C05428=1039.258,123.258,-94.133,169.875,39.736,157.485
C05429=1039.265,123.507,-94.154,169.877,39.737,157.486
C05430=1039.270,123.756,-94.175,169.879,39.737,157.486
C05431=1039.276,124.006,-94.195,169.881,39.737,157.486
C05432=1039.283,124.254,-94.216,169.883,39.738,157.486
C05433=1039.289,124.504,-94.237,169.886,39.738,157.486
C05434=1039.296,124.789,-94.260,169.888,39.739,157.486
C05435=1039.303,125.075,-94.284,169.891,39.739,157.487
C05436=1039.310,125.362,-94.307,169.893,39.740,157.487
C05437=1039.317,125.647,-94.331,169.895,39.740,157.487
C05438=1039.324,125.896,-94.352,169.897,39.741,157.487
C05439=1039.330,126.145,-94.372,169.899,39.741,157.487
C05440=1039.336,126.394,-94.393,169.902,39.741,157.487
C05441=1039.343,126.643,-94.414,169.905,39.741,157.487
C05442=1039.349,126.892,-94.434,169.907,39.742,157.488
C05443=1039.355,127.141,-94.456,169.909,39.742,157.488
C05444=1039.361,127.390,-94.476,169.911,39.743,157.488
C05445=1039.368,127.639,-94.497,169.913,39.743,157.488
C05446=1039.373,127.889,-94.517,169.915,39.744,157.488
C05447=1039.379,128.138,-94.537,169.918,39.744,157.488
C05448=1039.386,128.387,-94.558,169.920,39.745,157.489
C05449=1039.392,128.636,-94.579,169.922,39.744,157.489
C05450=1039.399,128.885,-94.600,169.924,39.745,157.489
C05451=1039.405,129.134,-94.620,169.926,39.745,157.489
C05452=1039.411,129.383,-94.642,169.928,39.746,157.489
C05453=1039.417,129.632,-94.662,169.930,39.746,157.489
C05454=1039.424,129.881,-94.683,169.934,39.747,157.490
C05455=1039.429,130.130,-94.704,169.936,39.747,157.490
C05456=1039.436,130.379,-94.725,169.938,39.748,157.490
C05457=1039.442,130.628,-94.746,169.940,39.747,157.490
C05458=1039.448,130.877,-94.766,169.942,39.748,157.490
C05459=1039.455,131.126,-94.787,169.944,39.748,157.490
C05460=1039.461,131.376,-94.808,169.946,39.749,157.490
C05461=1039.467,131.624,-94.829,169.948,39.749,157.491
C05462=1039.474,131.873,-94.850,169.951,39.750,157.491
C05463=1039.480,132.123,-94.871,169.953,39.750,157.491
C05464=1039.485,132.372,-94.893,169.955,39.751,157.491
C05465=1039.492,132.620,-94.914,169.957,39.752,157.491
C05466=1039.497,132.870,-94.934,169.959,39.752,157.492
C05467=1039.503,133.119,-94.956,169.963,39.753,157.492
C05468=1039.510,133.368,-94.977,169.965,39.753,157.492
C05469=1039.516,133.617,-94.998,169.967,39.753,157.492
C05470=1039.522,133.866,-95.019,169.969,39.754,157.492
C05471=1039.529,134.115,-95.040,169.971,39.754,157.492
C05472=1039.534,134.363,-95.061,169.973,39.755,157.493
C05473=1039.540,134.613,-95.082,169.975,39.755,157.493
C05474=1039.547,134.862,-95.103,169.978,39.756,157.493
C05475=1039.553,135.111,-95.125,169.980,39.756,157.493
C05476=1039.559,135.360,-95.146,169.982,39.757,157.493
C05477=1039.565,135.609,-95.167,169.984,39.757,157.493
C05478=1039.571,135.859,-95.188,169.986,39.758,157.494
C05479=1039.577,136.107,-95.210,169.988,39.758,157.494
C05480=1039.584,136.356,-95.231,169.992,39.758,157.494
C05481=1039.590,136.605,-95.252,169.994,39.759,157.494
C05482=1039.595,136.854,-95.273,169.996,39.759,157.494
C05483=1039.602,137.103,-95.294,169.998,39.760,157.494
C05484=1039.608,137.352,-95.315,170.000,39.760,157.495
C05485=1039.615,137.602,-95.337,170.002,39.761,157.495
C05486=1039.620,137.850,-95.358,170.005,39.761,157.495
C05487=1039.627,138.099,-95.379,170.007,39.762,157.495
C05488=1039.633,138.348,-95.401,170.009,39.762,157.495
C05489=1039.639,138.597,-95.423,170.011,39.763,157.496
C05490=1039.645,138.846,-95.443,170.014,39.764,157.496
C05491=1039.652,139.095,-95.464,170.016,39.764,157.496
C05492=1039.658,139.345,-95.486,170.019,39.764,157.496
C05493=1039.663,139.593,-95.507,170.021,39.765,157.496
C05494=1039.669,139.842,-95.529,170.023,39.765,157.497
C05495=1039.676,140.091,-95.550,170.025,39.766,157.497
C05496=1039.682,140.341,-95.572,170.027,39.766,157.497
C05497=1039.687,140.589,-95.593,170.029,39.767,157.497
C05498=1039.695,140.875,-95.618,170.033,39.768,157.497
C05499=1039.701,141.160,-95.642,170.035,39.768,157.498
C05500=1039.709,141.446,-95.668,170.037,39.769,157.498
C05501=1039.716,141.731,-95.692,170.040,39.770,157.498
C05502=1039.722,141.980,-95.714,170.042,39.770,157.498
C05503=1039.728,142.229,-95.735,170.045,39.771,157.498
C05504=1039.734,142.479,-95.757,170.047,39.771,157.499
C05505=1039.741,142.728,-95.779,170.049,39.772,157.499
C05506=1039.746,142.976,-95.800,170.051,39.772,157.499
C05507=1039.752,143.225,-95.821,170.054,39.772,157.499
C05508=1039.759,143.475,-95.843,170.057,39.773,157.499
C05509=1039.765,143.724,-95.865,170.059,39.774,157.500
C05510=1039.771,143.973,-95.886,170.061,39.774,157.500
C05511=1039.776,144.222,-95.908,170.063,39.775,157.500
C05512=1039.783,144.470,-95.930,170.065,39.775,157.500
C05513=1039.789,144.719,-95.952,170.067,39.776,157.500
C05514=1039.795,144.969,-95.973,170.070,39.776,157.500
C05515=1039.802,145.217,-95.994,170.073,39.777,157.501
C05516=1039.808,145.467,-96.016,170.075,39.778,157.501
C05517=1039.814,145.715,-96.037,170.077,39.778,157.501
C05518=1039.820,145.964,-96.059,170.079,39.779,157.501
C05519=1039.826,146.213,-96.081,170.081,39.779,157.501
C05520=1039.833,146.462,-96.103,170.084,39.780,157.502
C05521=1039.839,146.711,-96.124,170.087,39.780,157.502
C05522=1039.845,146.961,-96.146,170.089,39.780,157.502
C05523=1039.851,147.209,-96.168,170.091,39.781,157.502
C05524=1039.858,147.458,-96.190,170.093,39.782,157.502
C05525=1039.863,147.707,-96.211,170.095,39.782,157.503
C05526=1039.869,147.956,-96.234,170.098,39.783,157.503
C05527=1039.875,148.205,-96.256,170.100,39.783,157.503
C05528=1039.881,148.454,-96.278,170.103,39.784,157.503
C05529=1039.887,148.703,-96.299,170.105,39.785,157.503
C05530=1039.894,148.952,-96.322,170.107,39.785,157.504
C05531=1039.900,149.201,-96.343,170.110,39.786,157.504
C05532=1039.906,149.450,-96.365,170.112,39.787,157.504
C05533=1039.912,149.698,-96.387,170.114,39.787,157.504
C05534=1039.917,149.948,-96.409,170.117,39.788,157.504
C05535=1039.924,150.197,-96.431,170.119,39.788,157.505
C05536=1039.930,150.446,-96.453,170.122,39.789,157.505
C05537=1039.936,150.695,-96.475,170.124,39.790,157.505
C05538=1039.942,150.944,-96.496,170.126,39.790,157.505
C05539=1039.948,151.193,-96.519,170.128,39.790,157.505
C05540=1039.954,151.442,-96.541,170.131,39.791,157.506
C05541=1039.961,151.691,-96.563,170.134,39.792,157.506
C05542=1039.967,151.940,-96.585,170.136,39.792,157.506
C05543=1039.973,152.189,-96.607,170.138,39.793,157.506
C05544=1039.979,152.438,-96.629,170.140,39.794,157.506
C05545=1039.985,152.687,-96.652,170.142,39.794,157.507
C05546=1039.991,152.935,-96.673,170.145,39.795,157.507
C05547=1039.997,153.184,-96.695,170.148,39.795,157.507
C05548=1040.003,153.433,-96.717,170.150,39.796,157.507
C05549=1040.009,153.682,-96.740,170.152,39.797,157.507
C05550=1040.015,153.931,-96.762,170.154,39.797,157.508
C05551=1040.022,154.180,-96.784,170.157,39.798,157.508
C05552=1040.028,154.429,-96.806,170.160,39.799,157.508
C05553=1040.034,154.678,-96.829,170.162,39.799,157.508
C05554=1040.040,154.927,-96.850,170.164,39.800,157.508
C05555=1040.046,155.175,-96.873,170.166,39.801,157.509
C05556=1040.052,155.425,-96.895,170.169,39.801,157.509
C05557=1040.058,155.674,-96.917,170.172,39.801,157.509
C05558=1040.064,155.922,-96.940,170.174,39.803,157.509
C05559=1040.070,156.172,-96.962,170.176,39.803,157.510
C05560=1040.077,156.420,-96.984,170.178,39.803,157.510
C05561=1040.082,156.670,-97.006,170.181,39.804,157.510
C05562=1040.090,156.955,-97.032,170.184,39.805,157.510
C05563=1040.096,157.240,-97.057,170.187,39.806,157.511
C05564=1040.104,157.525,-97.083,170.189,39.806,157.511
C05565=1040.111,157.811,-97.109,170.192,39.807,157.511
C05566=1040.117,158.060,-97.131,170.195,39.808,157.511
C05567=1040.123,158.308,-97.154,170.197,39.808,157.511
C05568=1040.129,158.558,-97.176,170.199,39.809,157.512
C05569=1040.135,158.807,-97.199,170.202,39.810,157.512
C05570=1040.141,159.055,-97.221,170.204,39.810,157.512
C05571=1040.148,159.304,-97.243,170.207,39.811,157.512
C05572=1040.153,159.553,-97.266,170.209,39.812,157.513
C05573=1040.160,159.802,-97.288,170.212,39.812,157.513
C05574=1040.166,160.050,-97.310,170.214,39.813,157.513
C05575=1040.172,160.299,-97.333,170.216,39.814,157.513
C05576=1040.177,160.549,-97.355,170.219,39.815,157.514
C05577=1040.183,160.798,-97.378,170.221,39.815,157.514
C05578=1040.190,161.046,-97.401,170.224,39.816,157.514
C05579=1040.195,161.295,-97.424,170.226,39.817,157.514
C05580=1040.201,161.544,-97.447,170.229,39.818,157.514
C05581=1040.207,161.793,-97.470,170.231,39.819,157.515
C05582=1040.213,162.042,-97.492,170.233,39.819,157.515
C05583=1040.219,162.290,-97.515,170.236,39.820,157.515
C05584=1040.225,162.539,-97.538,170.239,39.821,157.515
C05585=1040.230,162.788,-97.561,170.241,39.822,157.516
C05586=1040.237,163.038,-97.584,170.243,39.822,157.516
C05587=1040.243,163.286,-97.606,170.245,39.823,157.516
C05588=1040.249,163.535,-97.629,170.248,39.824,157.516
C05589=1040.255,163.784,-97.652,170.251,39.825,157.517
C05590=1040.260,164.033,-97.675,170.253,39.826,157.517
C05591=1040.266,164.282,-97.698,170.255,39.826,157.517
C05592=1040.273,164.531,-97.721,170.259,39.827,157.518
C05593=1040.278,164.780,-97.743,170.261,39.828,157.518
C05594=1040.284,165.028,-97.766,170.263,39.829,157.518
C05595=1040.290,165.277,-97.789,170.265,39.829,157.518
C05596=1040.295,165.526,-97.812,170.267,39.830,157.518
C05597=1040.302,165.775,-97.835,170.271,39.831,157.519
C05598=1040.308,166.024,-97.858,170.273,39.832,157.519
C05599=1040.314,166.273,-97.881,170.275,39.833,157.519
C05600=1040.320,166.522,-97.904,170.277,39.833,157.519
C05601=1040.325,166.771,-97.927,170.281,39.834,157.520
C05602=1040.332,167.020,-97.949,170.283,39.835,157.520
C05603=1040.338,167.269,-97.972,170.285,39.836,157.520
C05604=1040.344,167.517,-97.996,170.288,39.837,157.521
C05605=1040.350,167.766,-98.019,170.291,39.837,157.521
C05606=1040.356,168.015,-98.042,170.293,39.838,157.521
C05607=1040.362,168.264,-98.064,170.295,39.839,157.521
C05608=1040.368,168.513,-98.087,170.298,39.840,157.522
C05609=1040.374,168.762,-98.110,170.301,39.841,157.522
C05610=1040.380,169.010,-98.134,170.303,39.841,157.522
C05611=1040.386,169.260,-98.157,170.305,39.842,157.522
C05612=1040.392,169.509,-98.180,170.308,39.843,157.522
C05613=1040.398,169.757,-98.203,170.311,39.844,157.523
C05614=1040.404,170.006,-98.225,170.313,39.844,157.523
C05615=1040.411,170.255,-98.250,170.316,39.845,157.523
C05616=1040.416,170.504,-98.272,170.318,39.846,157.524
C05617=1040.422,170.753,-98.295,170.320,39.847,157.524
C05618=1040.428,171.002,-98.318,170.324,39.848,157.524
C05619=1040.435,171.250,-98.341,170.326,39.848,157.524
C05620=1040.441,171.499,-98.365,170.328,39.849,157.525
C05621=1040.447,171.748,-98.388,170.330,39.850,157.525
C05622=1040.453,171.996,-98.411,170.334,39.851,157.525
C05623=1040.458,172.245,-98.434,170.336,39.852,157.525
C05624=1040.465,172.495,-98.458,170.338,39.852,157.526
C05625=1040.471,172.744,-98.481,170.341,39.853,157.526
C05626=1040.478,173.028,-98.507,170.344,39.854,157.526
C05627=1040.484,173.313,-98.534,170.347,39.855,157.526
C05628=1040.492,173.598,-98.560,170.350,39.856,157.527
C05629=1040.499,173.883,-98.587,170.352,39.857,157.527
C05630=1040.505,174.131,-98.611,170.356,39.858,157.527
C05631=1040.511,174.380,-98.633,170.358,39.859,157.528
C05632=1040.518,174.630,-98.656,170.360,39.859,157.528
C05633=1040.524,174.878,-98.680,170.364,39.860,157.528
C05634=1040.530,175.127,-98.703,170.366,39.861,157.528
C05635=1040.536,175.376,-98.727,170.369,39.862,157.529
C05636=1040.542,175.625,-98.750,170.371,39.863,157.529
C05637=1040.548,175.873,-98.774,170.373,39.863,157.529
C05638=1040.554,176.122,-98.797,170.377,39.864,157.529
C05639=1040.561,176.371,-98.819,170.379,39.865,157.530
C05640=1040.567,176.619,-98.843,170.381,39.866,157.530
C05641=1040.573,176.869,-98.866,170.385,39.867,157.530
C05642=1040.579,177.117,-98.890,170.387,39.867,157.530
C05643=1040.586,177.367,-98.913,170.390,39.868,157.531
C05644=1040.592,177.615,-98.937,170.392,39.869,157.531
C05645=1040.597,177.864,-98.960,170.394,39.870,157.531
C05646=1040.604,178.113,-98.984,170.398,39.871,157.531
C05647=1040.610,178.361,-99.007,170.400,39.872,157.532
C05648=1040.617,178.611,-99.030,170.403,39.872,157.532
C05649=1040.623,178.859,-99.054,170.406,39.873,157.532
C05650=1040.629,179.108,-99.077,170.408,39.874,157.533
C05651=1040.635,179.357,-99.101,170.411,39.875,157.533
C05652=1040.641,179.606,-99.124,170.413,39.876,157.533
C05653=1040.648,179.855,-99.148,170.417,39.877,157.533
C05654=1040.654,180.103,-99.171,170.419,39.877,157.534
C05655=1040.660,180.352,-99.195,170.421,39.878,157.534
C05656=1040.666,180.601,-99.218,170.424,39.878,157.534
C05657=1040.673,180.850,-99.242,170.427,39.880,157.534
C05658=1040.679,181.099,-99.265,170.430,39.881,157.535
C05659=1040.686,181.347,-99.289,170.432,39.881,157.535
C05660=1040.692,181.596,-99.312,170.435,39.882,157.535
C05661=1040.698,181.845,-99.336,170.438,39.883,157.536
C05662=1040.704,182.093,-99.359,170.440,39.883,157.536
C05663=1040.711,182.343,-99.383,170.443,39.884,157.536
C05664=1040.717,182.591,-99.406,170.445,39.886,157.536
C05665=1040.723,182.840,-99.430,170.449,39.887,157.537
C05666=1040.729,183.089,-99.454,170.451,39.887,157.537
C05667=1040.736,183.338,-99.477,170.454,39.888,157.537
C05668=1040.742,183.586,-99.501,170.456,39.889,157.537
C05669=1040.748,183.835,-99.525,170.460,39.890,157.538
C05670=1040.754,184.084,-99.549,170.462,39.891,157.538
C05671=1040.760,184.333,-99.573,170.464,39.892,157.538
C05672=1040.766,184.582,-99.598,170.468,39.893,157.539
C05673=1040.772,184.831,-99.622,170.470,39.894,157.539
C05674=1040.778,185.079,-99.646,170.473,39.895,157.539
C05675=1040.784,185.327,-99.670,170.475,39.896,157.539
C05676=1040.790,185.577,-99.694,170.478,39.897,157.540
C05677=1040.796,185.825,-99.718,170.481,39.898,157.540
C05678=1040.802,186.074,-99.742,170.483,39.899,157.540
C05679=1040.808,186.323,-99.766,170.487,39.900,157.541
C05680=1040.814,186.571,-99.790,170.489,39.901,157.541
C05681=1040.819,186.820,-99.814,170.491,39.902,157.541
C05682=1040.826,187.069,-99.838,170.495,39.903,157.542
C05683=1040.831,187.318,-99.863,170.497,39.905,157.542
C05684=1040.838,187.567,-99.887,170.500,39.906,157.542
C05685=1040.843,187.815,-99.911,170.503,39.907,157.543
C05686=1040.850,188.064,-99.935,170.506,39.908,157.543
C05687=1040.855,188.313,-99.959,170.508,39.909,157.543
C05688=1040.862,188.562,-99.983,170.511,39.910,157.544
C05689=1040.867,188.810,-100.008,170.514,39.911,157.544
C05690=1040.875,189.095,-100.036,170.517,39.912,157.544
C05691=1040.882,189.379,-100.063,170.520,39.913,157.545
C05692=1040.889,189.664,-100.091,170.523,39.914,157.545
C05693=1040.895,189.948,-100.119,170.526,39.915,157.545
C05694=1040.901,190.197,-100.143,170.530,39.916,157.546
C05695=1040.907,190.446,-100.167,170.532,39.917,157.546
C05696=1040.914,190.694,-100.192,170.535,39.918,157.546
C05697=1040.919,190.943,-100.216,170.537,39.919,157.547
C05698=1040.925,191.192,-100.240,170.541,39.920,157.547
C05699=1040.931,191.441,-100.265,170.543,39.921,157.547
C05700=1040.938,191.690,-100.289,170.546,39.922,157.548
C05701=1040.944,191.938,-100.314,170.549,39.923,157.548
C05702=1040.950,192.187,-100.338,170.551,39.925,157.548
C05703=1040.956,192.435,-100.362,170.554,39.926,157.549
C05704=1040.962,192.684,-100.386,170.557,39.927,157.549
C05705=1040.968,192.933,-100.411,170.560,39.928,157.549
C05706=1040.974,193.181,-100.435,170.563,39.929,157.550
C05707=1040.980,193.431,-100.460,170.566,39.930,157.550
C05708=1040.987,193.679,-100.484,170.569,39.931,157.550
C05709=1040.993,193.928,-100.509,170.571,39.932,157.551
C05710=1040.999,194.177,-100.533,170.575,39.933,157.551
C05711=1041.005,194.425,-100.558,170.577,39.934,157.551
C05712=1041.011,194.674,-100.582,170.580,39.935,157.552
C05713=1041.017,194.923,-100.606,170.582,39.936,157.552
C05714=1041.024,195.171,-100.632,170.586,39.938,157.552
C05715=1041.030,195.420,-100.656,170.588,39.939,157.553
C05716=1041.036,195.669,-100.680,170.592,39.940,157.553
C05717=1041.042,195.917,-100.705,170.594,39.941,157.553
C05718=1041.048,196.167,-100.729,170.597,39.942,157.554
C05719=1041.055,196.415,-100.754,170.599,39.943,157.554
C05720=1041.061,196.664,-100.778,170.603,39.944,157.554
C05721=1041.067,196.912,-100.804,170.606,39.945,157.555
C05722=1041.073,197.161,-100.828,170.608,39.946,157.555
C05723=1041.079,197.411,-100.852,170.612,39.948,157.555
C05724=1041.086,197.658,-100.877,170.614,39.949,157.556
C05725=1041.092,197.907,-100.901,170.617,39.950,157.556
C05726=1041.099,198.156,-100.926,170.620,39.951,157.556
C05727=1041.104,198.405,-100.951,170.623,39.952,157.557
C05728=1041.111,198.654,-100.976,170.626,39.953,157.557
C05729=1041.117,198.902,-101.000,170.629,39.954,157.557
C05730=1041.123,199.151,-101.025,170.632,39.955,157.558
C05731=1041.130,199.399,-101.050,170.634,39.956,157.558
C05732=1041.136,199.648,-101.074,170.638,39.957,157.558
C05733=1041.142,199.897,-101.100,170.641,39.958,157.559
C05734=1041.148,200.145,-101.123,170.643,39.959,157.559
C05735=1041.154,200.394,-101.149,170.647,39.961,157.559
C05736=1041.161,200.643,-101.173,170.649,39.962,157.560
C05737=1041.167,200.892,-101.198,170.652,39.963,157.560
C05738=1041.173,201.140,-101.223,170.656,39.964,157.560
C05739=1041.180,201.389,-101.247,170.658,39.966,157.561
C05740=1041.186,201.638,-101.273,170.661,39.967,157.561
C05741=1041.192,201.886,-101.298,170.664,39.968,157.561
C05742=1041.198,202.135,-101.323,170.667,39.969,157.562
C05743=1041.204,202.384,-101.348,170.670,39.970,157.562
C05744=1041.210,202.633,-101.373,170.673,39.971,157.563
C05745=1041.216,202.881,-101.398,170.676,39.973,157.563
C05746=1041.222,203.130,-101.424,170.679,39.974,157.563
C05747=1041.228,203.378,-101.448,170.682,39.975,157.564
C05748=1041.234,203.627,-101.473,170.684,39.977,157.564
C05749=1041.240,203.876,-101.499,170.688,39.978,157.564
C05750=1041.246,204.124,-101.524,170.691,39.979,157.565
C05751=1041.253,204.373,-101.549,170.693,39.980,157.565
C05752=1041.259,204.622,-101.574,170.697,39.982,157.566
C05753=1041.266,204.870,-101.599,170.700,39.983,157.566
C05754=1041.292,205.922,-101.705,170.981,40.086,157.599
C05755=1041.299,206.221,-101.737,170.984,40.088,157.599
C05756=1041.308,206.520,-101.769,170.986,40.091,157.600
C05757=1041.316,206.820,-101.801,170.989,40.093,157.600
C05758=1041.324,207.120,-101.833,170.992,40.095,157.601
C05759=1041.330,207.369,-101.859,170.994,40.097,157.601
C05760=1041.337,207.617,-101.886,170.996,40.099,157.602
C05761=1041.344,207.865,-101.912,170.998,40.101,157.602
C05762=1041.351,208.114,-101.938,171.001,40.104,157.603
C05763=1041.356,208.362,-101.965,171.002,40.105,157.603
C05764=1041.364,208.611,-101.991,171.005,40.108,157.604
C05765=1041.371,208.860,-102.018,171.007,40.109,157.605
C05766=1041.376,209.108,-102.044,171.009,40.112,157.605
C05767=1041.384,209.357,-102.071,171.011,40.113,157.606
C05768=1041.390,209.605,-102.097,171.014,40.116,157.606
C05769=1041.397,209.854,-102.124,171.015,40.117,157.607
C05770=1041.403,210.102,-102.150,171.018,40.120,157.607
C05771=1041.410,210.350,-102.177,171.021,40.121,157.608
C05772=1041.417,210.599,-102.204,171.023,40.124,157.608
C05773=1041.423,210.847,-102.230,171.025,40.125,157.609
C05774=1041.430,211.097,-102.257,171.027,40.128,157.609
C05775=1041.437,211.345,-102.284,171.030,40.129,157.610
C05776=1041.444,211.593,-102.310,171.031,40.132,157.610
C05777=1041.450,211.842,-102.337,171.034,40.133,157.611
C05778=1041.456,212.090,-102.363,171.036,40.136,157.611
C05779=1041.463,212.339,-102.390,171.038,40.137,157.612
C05780=1041.470,212.587,-102.417,171.040,40.140,157.612
C05781=1041.476,212.835,-102.444,171.043,40.141,157.613
C05782=1041.482,213.084,-102.471,171.045,40.144,157.613
C05783=1041.489,213.332,-102.498,171.047,40.146,157.614
C05784=1041.496,213.581,-102.525,171.050,40.148,157.614
C05785=1041.503,213.830,-102.551,171.052,40.150,157.615
C05786=1041.509,214.077,-102.579,171.054,40.152,157.615
C05787=1041.516,214.326,-102.605,171.056,40.154,157.616
C05788=1041.522,214.575,-102.632,171.059,40.156,157.616
C05789=1041.529,214.823,-102.659,171.061,40.158,157.617
C05790=1041.535,215.072,-102.686,171.063,40.160,157.617
C05791=1041.542,215.321,-102.713,171.065,40.162,157.618
C05792=1041.549,215.568,-102.740,171.068,40.164,157.618
C05793=1041.555,215.817,-102.767,171.070,40.166,157.619
C05794=1041.562,216.066,-102.793,171.072,40.168,157.619
C05795=1041.568,216.314,-102.820,171.074,40.170,157.620
C05796=1041.575,216.563,-102.847,171.077,40.172,157.620
C05797=1041.582,216.811,-102.875,171.080,40.174,157.621
C05798=1041.588,217.060,-102.902,171.081,40.176,157.621
C05799=1041.595,217.308,-102.928,171.084,40.178,157.622
C05800=1041.602,217.557,-102.955,171.086,40.179,157.622
C05801=1041.609,217.805,-102.982,171.089,40.182,157.623
C05802=1041.615,218.053,-103.009,171.090,40.183,157.623
C05803=1041.622,218.302,-103.036,171.093,40.186,157.624
C05804=1041.629,218.550,-103.063,171.095,40.187,157.624
C05805=1041.635,218.799,-103.090,171.098,40.190,157.625
C05806=1041.642,219.047,-103.117,171.100,40.191,157.626
C05807=1041.648,219.296,-103.144,171.102,40.194,157.626
C05808=1041.656,219.544,-103.171,171.104,40.195,157.627
C05809=1041.662,219.793,-103.198,171.107,40.198,157.627
C05810=1041.669,220.041,-103.226,171.109,40.199,157.628
C05811=1041.677,220.346,-103.259,171.112,40.202,157.628
C05812=1041.685,220.651,-103.292,171.115,40.204,157.629
C05813=1041.692,220.956,-103.326,171.117,40.207,157.629
C05814=1041.701,221.262,-103.360,171.121,40.209,157.630
C05815=1041.707,221.510,-103.386,171.123,40.211,157.631
C05816=1041.713,221.758,-103.414,171.125,40.213,157.631
C05817=1041.721,222.007,-103.441,171.128,40.216,157.632
C05818=1041.727,222.255,-103.469,171.130,40.217,157.632
C05819=1041.734,222.504,-103.496,171.133,40.220,157.633
C05820=1041.740,222.752,-103.523,171.134,40.221,157.633
C05821=1041.747,223.000,-103.551,171.137,40.224,157.634
C05822=1041.753,223.249,-103.578,171.140,40.225,157.634
C05823=1041.760,223.497,-103.605,171.142,40.228,157.635
C05824=1041.767,223.746,-103.633,171.145,40.229,157.635
C05825=1041.773,223.994,-103.660,171.147,40.231,157.636
C05826=1041.780,224.243,-103.687,171.150,40.234,157.637
C05827=1041.786,224.491,-103.715,171.151,40.235,157.637
C05828=1041.793,224.740,-103.743,171.154,40.238,157.638
C05829=1041.800,224.988,-103.771,171.156,40.239,157.638
C05830=1041.806,225.236,-103.798,171.159,40.242,157.639
C05831=1041.813,225.485,-103.824,171.162,40.243,157.639
C05832=1041.819,225.733,-103.852,171.164,40.246,157.640
C05833=1041.826,225.981,-103.880,171.167,40.247,157.640
C05834=1041.833,226.230,-103.908,171.168,40.250,157.641
C05835=1041.840,226.478,-103.935,171.171,40.251,157.641
C05836=1041.846,226.727,-103.963,171.173,40.253,157.642
C05837=1041.853,226.976,-103.990,171.176,40.255,157.642
C05838=1041.859,227.224,-104.018,171.178,40.257,157.643
C05839=1041.867,227.472,-104.045,171.181,40.259,157.643
C05840=1041.873,227.720,-104.072,171.183,40.261,157.644
C05841=1041.879,227.969,-104.100,171.186,40.263,157.644
C05842=1041.886,228.217,-104.128,171.189,40.265,157.645
C05843=1041.893,228.465,-104.155,171.190,40.267,157.645
C05844=1041.899,228.714,-104.183,171.193,40.269,157.646
C05845=1041.906,228.962,-104.211,171.195,40.271,157.646
C05846=1041.913,229.211,-104.239,171.198,40.273,157.647
C05847=1041.920,229.459,-104.266,171.200,40.275,157.647
C05848=1041.926,229.708,-104.294,171.203,40.277,157.648
C05849=1041.932,229.956,-104.322,171.205,40.279,157.648
C05850=1041.939,230.205,-104.350,171.208,40.281,157.649
C05851=1041.946,230.453,-104.378,171.211,40.283,157.650
C05852=1041.952,230.701,-104.405,171.213,40.285,157.650
C05853=1041.958,230.949,-104.433,171.215,40.287,157.651
C05854=1041.965,231.198,-104.461,171.217,40.289,157.651
C05855=1041.972,231.446,-104.489,171.220,40.291,157.652
C05856=1041.979,231.694,-104.517,171.222,40.293,157.652
C05857=1041.985,231.943,-104.545,171.225,40.295,157.653
C05858=1041.991,232.191,-104.573,171.227,40.297,157.653
C05859=1041.998,232.440,-104.601,171.230,40.299,157.654
C05860=1042.005,232.688,-104.628,171.233,40.301,157.654
C05861=1042.012,232.936,-104.657,171.235,40.303,157.655
C05862=1042.018,233.185,-104.685,171.238,40.305,157.655
C05863=1042.024,233.433,-104.713,171.240,40.307,157.656
C05864=1042.031,233.682,-104.741,171.243,40.309,157.657
C05865=1042.038,233.930,-104.768,171.246,40.312,157.657
C05866=1042.044,234.178,-104.797,171.248,40.313,157.658
C05867=1042.052,234.476,-104.831,171.251,40.316,157.658
C05868=1042.060,234.774,-104.864,171.253,40.318,157.659
C05869=1042.068,235.071,-104.898,171.257,40.321,157.659
C05870=1042.076,235.369,-104.932,171.260,40.323,157.660
C05871=1042.082,235.618,-104.960,171.262,40.325,157.661
C05872=1042.089,235.866,-104.988,171.265,40.327,157.661
C05873=1042.096,236.114,-105.016,171.267,40.329,157.662
C05874=1042.102,236.362,-105.044,171.270,40.331,157.662
C05875=1042.108,236.611,-105.072,171.273,40.333,157.663
C05876=1042.115,236.859,-105.101,171.275,40.335,157.663
C05877=1042.122,237.107,-105.129,171.278,40.337,157.664
C05878=1042.128,237.355,-105.158,171.280,40.339,157.664
C05879=1042.135,237.604,-105.185,171.283,40.341,157.665
C05880=1042.142,237.852,-105.213,171.286,40.343,157.666
C05881=1042.149,238.100,-105.242,171.288,40.345,157.666
C05882=1042.155,238.349,-105.270,171.291,40.347,157.667
C05883=1042.162,238.597,-105.298,171.293,40.349,157.667
C05884=1042.168,238.845,-105.326,171.296,40.351,157.668
C05885=1042.175,239.094,-105.355,171.298,40.353,157.668
C05886=1042.182,239.342,-105.383,171.301,40.355,157.669
C05887=1042.188,239.591,-105.412,171.303,40.357,157.669
C05888=1042.195,239.839,-105.440,171.306,40.359,157.670
C05889=1042.202,240.087,-105.468,171.309,40.361,157.670
C05890=1042.208,240.336,-105.497,171.311,40.363,157.671
C05891=1042.215,240.583,-105.525,171.314,40.365,157.671
C05892=1042.221,240.832,-105.553,171.316,40.367,157.672
C05893=1042.228,241.081,-105.582,171.319,40.369,157.672
C05894=1042.235,241.329,-105.610,171.322,40.371,157.673
C05895=1042.241,241.577,-105.639,171.325,40.373,157.674
C05896=1042.248,241.825,-105.667,171.328,40.376,157.674
C05897=1042.254,242.074,-105.696,171.330,40.377,157.675
C05898=1042.260,242.322,-105.725,171.333,40.379,157.675
C05899=1042.267,242.570,-105.753,171.335,40.382,157.676
C05900=1042.273,242.819,-105.782,171.338,40.383,157.676
C05901=1042.281,243.067,-105.810,171.341,40.385,157.677
C05902=1042.287,243.315,-105.839,171.343,40.388,157.678
C05903=1042.293,243.563,-105.869,171.346,40.389,157.678
C05904=1042.300,243.812,-105.896,171.348,40.392,157.679
C05905=1042.306,244.060,-105.925,171.351,40.394,157.679
C05906=1042.313,244.308,-105.954,171.354,40.396,157.680
C05907=1042.320,244.557,-105.983,171.356,40.398,157.680
C05908=1042.326,244.805,-106.011,171.359,40.400,157.681
C05909=1042.333,245.053,-106.040,171.361,40.402,157.681
C05910=1042.339,245.301,-106.069,171.365,40.404,157.682
C05911=1042.345,245.549,-106.098,171.367,40.406,157.683
C05912=1042.352,245.797,-106.126,171.370,40.408,157.683
C05913=1042.359,246.046,-106.156,171.373,40.410,157.684
C05914=1042.366,246.294,-106.185,171.375,40.412,157.684
C05915=1042.372,246.542,-106.214,171.378,40.414,157.685
C05916=1042.378,246.791,-106.242,171.380,40.416,157.685
C05917=1042.384,247.039,-106.271,171.383,40.419,157.686
C05918=1042.390,247.287,-106.300,171.386,40.421,157.687
C05919=1042.398,247.536,-106.329,171.388,40.423,157.687
C05920=1042.404,247.784,-106.358,171.391,40.425,157.688
C05921=1042.410,248.032,-106.387,171.393,40.427,157.688
C05922=1042.417,248.280,-106.416,171.397,40.429,157.689
C05923=1042.424,248.572,-106.451,171.400,40.431,157.689
C05924=1042.432,248.864,-106.485,171.404,40.434,157.690
C05925=1042.440,249.156,-106.519,171.406,40.436,157.691
C05926=1042.448,249.448,-106.553,171.410,40.439,157.692
C05927=1042.454,249.696,-106.582,171.413,40.441,157.692
C05928=1042.460,249.944,-106.611,171.415,40.443,157.693
C05929=1042.467,250.192,-106.640,171.418,40.445,157.693
C05930=1042.473,250.441,-106.670,171.420,40.447,157.694
C05931=1042.480,250.689,-106.699,171.423,40.450,157.694
C05932=1042.486,250.937,-106.729,171.426,40.451,157.695
C05933=1042.493,251.184,-106.757,171.429,40.453,157.695
C05934=1042.500,251.433,-106.786,171.432,40.456,157.696
C05935=1042.506,251.681,-106.815,171.434,40.458,157.697
C05936=1042.513,251.930,-106.845,171.437,40.459,157.697
C05937=1042.519,252.178,-106.874,171.440,40.462,157.698
C05938=1042.526,252.427,-106.903,171.442,40.464,157.698
C05939=1042.532,252.674,-106.933,171.446,40.466,157.699
C05940=1042.539,252.923,-106.962,171.449,40.468,157.700
C05941=1042.545,253.171,-106.991,171.451,40.470,157.700
C05942=1042.552,253.419,-107.020,171.454,40.472,157.701
C05943=1042.560,253.667,-107.050,171.456,40.474,157.701
C05944=1042.566,253.915,-107.079,171.460,40.476,157.702
C05945=1042.572,254.163,-107.108,171.462,40.478,157.702
C05946=1042.579,254.412,-107.137,171.465,40.480,157.703
C05947=1042.585,254.660,-107.167,171.468,40.483,157.703
C05948=1042.592,254.908,-107.196,171.470,40.485,157.704
C05949=1042.599,255.157,-107.225,171.474,40.487,157.705
C05950=1042.605,255.404,-107.255,171.477,40.488,157.705
C05951=1042.612,255.653,-107.285,171.479,40.491,157.706
C05952=1042.618,255.901,-107.314,171.482,40.493,157.706
C05953=1042.625,256.149,-107.344,171.485,40.495,157.707
C05954=1042.632,256.397,-107.372,171.488,40.497,157.707
C05955=1042.639,256.646,-107.402,171.491,40.499,157.708
C05956=1042.646,256.893,-107.431,171.493,40.501,157.709
C05957=1042.652,257.142,-107.460,171.497,40.503,157.709
C05958=1042.659,257.390,-107.491,171.500,40.505,157.710
C05959=1042.665,257.638,-107.520,171.502,40.507,157.710
C05960=1042.672,257.887,-107.549,171.505,40.509,157.711
C05961=1042.679,258.134,-107.579,171.508,40.511,157.712
C05962=1042.686,258.383,-107.608,171.511,40.514,157.712
C05963=1042.692,258.631,-107.638,171.513,40.515,157.713
C05964=1042.699,258.879,-107.667,171.517,40.517,157.713
C05965=1042.706,259.127,-107.697,171.520,40.520,157.714
C05966=1042.712,259.376,-107.726,171.522,40.522,157.714
C05967=1042.719,259.623,-107.756,171.525,40.524,157.715
C05968=1042.726,259.872,-107.786,171.529,40.525,157.716
C05969=1042.733,260.119,-107.815,171.531,40.528,157.716
C05970=1042.740,260.368,-107.844,171.534,40.530,157.717
C05971=1042.747,260.616,-107.874,171.537,40.532,157.717
C05972=1042.754,260.864,-107.904,171.540,40.534,157.718
C05973=1042.761,261.113,-107.933,171.543,40.536,157.718
C05974=1042.767,261.360,-107.963,171.546,40.538,157.719
C05975=1042.774,261.609,-107.993,171.549,40.540,157.720
C05976=1042.781,261.857,-108.022,171.552,40.542,157.720
C05977=1042.788,262.105,-108.052,171.555,40.544,157.721
C05978=1042.795,262.354,-108.082,171.558,40.546,157.721
C05979=1042.802,262.644,-108.118,171.562,40.549,157.722
C05980=1042.810,262.934,-108.152,171.564,40.551,157.723
C05981=1042.817,263.224,-108.187,171.568,40.554,157.723
C05982=1042.825,263.515,-108.222,171.572,40.556,157.724
C05983=1042.832,263.763,-108.252,171.574,40.559,157.725
C05984=1042.838,264.011,-108.283,171.577,40.561,157.725
C05985=1042.845,264.259,-108.313,171.581,40.563,157.726
C05986=1042.851,264.507,-108.343,171.583,40.565,157.727
C05987=1042.858,264.755,-108.373,171.586,40.567,157.727
C05988=1042.864,265.004,-108.403,171.590,40.569,157.728
C05989=1042.871,265.252,-108.433,171.592,40.571,157.728
C05990=1042.878,265.500,-108.463,171.595,40.573,157.729
C05991=1042.884,265.748,-108.493,171.599,40.575,157.730
C05992=1042.891,265.996,-108.523,171.601,40.578,157.730
C05993=1042.898,266.244,-108.553,171.604,40.580,157.731
C05994=1042.904,266.492,-108.584,171.608,40.582,157.731
C05995=1042.911,266.740,-108.614,171.610,40.584,157.732
C05996=1042.918,266.989,-108.644,171.614,40.586,157.733
C05997=1042.924,267.236,-108.674,171.617,40.588,157.733
C05998=1042.931,267.484,-108.704,171.619,40.591,157.734
C05999=1042.937,267.732,-108.735,171.623,40.593,157.734
C06000=1042.944,267.980,-108.765,171.625,40.595,157.735
C06001=1042.951,268.229,-108.796,171.628,40.597,157.736
C06002=1042.957,268.476,-108.825,171.632,40.599,157.736
C06003=1042.964,268.725,-108.856,171.634,40.601,157.737
C06004=1042.971,268.973,-108.886,171.638,40.604,157.738
C06005=1042.977,269.221,-108.916,171.641,40.606,157.738
C06006=1042.984,269.469,-108.947,171.643,40.608,157.739
C06007=1042.991,269.717,-108.978,171.647,40.610,157.739
C06008=1042.997,269.965,-109.008,171.650,40.612,157.740
C06009=1043.004,270.213,-109.038,171.653,40.614,157.741
C06010=1043.011,270.461,-109.069,171.656,40.617,157.741
C06011=1043.017,270.709,-109.099,171.659,40.619,157.742
C06012=1043.024,270.957,-109.130,171.662,40.621,157.742
C06013=1043.030,271.205,-109.161,171.665,40.623,157.743
C06014=1043.038,271.453,-109.191,171.669,40.626,157.744
C06015=1043.043,271.701,-109.221,171.672,40.628,157.744
C06016=1043.051,271.949,-109.252,171.675,40.630,157.745
C06017=1043.057,272.197,-109.283,171.678,40.632,157.746
C06018=1043.064,272.446,-109.313,171.681,40.634,157.746
C06019=1043.071,272.693,-109.344,171.684,40.637,157.747
C06020=1043.077,272.941,-109.374,171.687,40.639,157.747
C06021=1043.083,273.190,-109.405,171.690,40.641,157.748
C06022=1043.090,273.437,-109.436,171.693,40.643,157.749
C06023=1043.097,273.685,-109.466,171.697,40.646,157.749
C06024=1043.103,273.934,-109.497,171.700,40.648,157.750
C06025=1043.111,274.181,-109.528,171.703,40.650,157.751
C06026=1043.117,274.430,-109.559,171.706,40.652,157.751
C06027=1043.123,274.677,-109.590,171.710,40.654,157.752
C06028=1043.130,274.925,-109.620,171.712,40.657,157.753
C06029=1043.137,275.173,-109.651,171.715,40.659,157.753
C06030=1043.143,275.422,-109.682,171.719,40.661,157.754
C06031=1043.150,275.669,-109.713,171.721,40.664,157.755
C06032=1043.157,275.917,-109.743,171.725,40.666,157.755
C06033=1043.163,276.165,-109.775,171.728,40.668,157.756
C06034=1043.170,276.414,-109.805,171.731,40.670,157.756
C06035=1043.178,276.708,-109.842,171.735,40.673,157.757
C06036=1043.186,277.003,-109.879,171.739,40.675,157.758
C06037=1043.194,277.298,-109.915,171.743,40.678,157.759
C06038=1043.202,277.593,-109.952,171.747,40.681,157.759
C06039=1043.208,277.840,-109.983,171.749,40.683,157.760
C06040=1043.215,278.089,-110.014,171.753,40.686,157.761
C06041=1043.222,278.337,-110.046,171.756,40.688,157.761
C06042=1043.229,278.584,-110.076,171.760,40.690,157.762
C06043=1043.235,278.833,-110.107,171.762,40.692,157.763
C06044=1043.242,279.081,-110.139,171.766,40.694,157.763
C06045=1043.249,279.329,-110.170,171.769,40.697,157.764
C06046=1043.255,279.577,-110.200,171.772,40.699,157.765
C06047=1043.261,279.824,-110.232,171.776,40.701,157.765
C06048=1043.268,280.072,-110.263,171.779,40.704,157.766
C06049=1043.275,280.320,-110.295,171.783,40.706,157.767
C06050=1043.282,280.568,-110.326,171.785,40.708,157.767
C06051=1043.288,280.817,-110.357,171.789,40.711,157.768
C06052=1043.295,281.065,-110.388,171.792,40.713,157.769
C06053=1043.302,281.313,-110.420,171.795,40.715,157.769
C06054=1043.308,281.560,-110.451,171.798,40.718,157.770
C06055=1043.314,281.808,-110.482,171.802,40.720,157.771
C06056=1043.321,282.056,-110.514,171.805,40.722,157.771
C06057=1043.328,282.303,-110.545,171.808,40.724,157.772
C06058=1043.335,282.551,-110.577,171.812,40.727,157.773
C06059=1043.341,282.799,-110.608,171.815,40.729,157.773
C06060=1043.348,283.047,-110.639,171.819,40.732,157.774
C06061=1043.355,283.295,-110.671,171.821,40.734,157.775
C06062=1043.361,283.543,-110.702,171.825,40.736,157.775
C06063=1043.368,283.791,-110.734,171.828,40.739,157.776
C06064=1043.375,284.039,-110.765,171.832,40.741,157.777
C06065=1043.382,284.287,-110.797,171.835,40.743,157.777
C06066=1043.388,284.535,-110.828,171.838,40.746,157.778
C06067=1043.395,284.782,-110.859,171.842,40.748,157.779
C06068=1043.402,285.030,-110.891,171.845,40.750,157.779
C06069=1043.409,285.278,-110.922,171.848,40.753,157.780
C06070=1043.415,285.526,-110.954,171.852,40.755,157.781
C06071=1043.422,285.774,-110.985,171.855,40.757,157.781
C06072=1043.429,286.022,-111.017,171.858,40.760,157.782
C06073=1043.435,286.270,-111.048,171.862,40.762,157.783
C06074=1043.443,286.518,-111.080,171.865,40.764,157.784
C06075=1043.449,286.767,-111.112,171.869,40.767,157.784
C06076=1043.456,287.014,-111.144,171.872,40.769,157.785
C06077=1043.462,287.262,-111.175,171.875,40.771,157.786
C06078=1043.469,287.510,-111.207,171.879,40.773,157.786
C06079=1043.476,287.758,-111.238,171.883,40.776,157.787
C06080=1043.483,288.005,-111.270,171.885,40.778,157.788
C06081=1043.489,288.253,-111.302,171.889,40.781,157.788
C06082=1043.496,288.501,-111.334,171.893,40.783,157.789
C06083=1043.503,288.748,-111.366,171.896,40.786,157.790
C06084=1043.509,288.996,-111.397,171.899,40.788,157.790
C06085=1043.516,289.245,-111.430,171.902,40.791,157.791
C06086=1043.523,289.492,-111.462,171.906,40.793,157.792
C06087=1043.530,289.740,-111.493,171.910,40.795,157.793
C06088=1043.536,289.988,-111.525,171.913,40.797,157.793
C06089=1043.543,290.236,-111.558,171.916,40.800,157.794
C06090=1043.550,290.484,-111.589,171.920,40.802,157.795
C06091=1043.558,290.790,-111.629,171.924,40.806,157.796
C06092=1043.567,291.097,-111.668,171.929,40.809,157.797
C06093=1043.574,291.403,-111.708,171.933,40.811,157.797
C06094=1043.583,291.710,-111.748,171.937,40.815,157.798
C06095=1043.590,291.958,-111.780,171.940,40.817,157.799
C06096=1043.596,292.206,-111.812,171.944,40.819,157.800
C06097=1043.603,292.454,-111.844,171.947,40.822,157.800
C06098=1043.610,292.702,-111.876,171.951,40.824,157.801
C06099=1043.616,292.949,-111.908,171.955,40.827,157.802
C06100=1043.623,293.197,-111.940,171.958,40.829,157.802
C06101=1043.631,293.445,-111.972,171.961,40.832,157.803
C06102=1043.637,293.693,-112.005,171.965,40.834,157.804
C06103=1043.644,293.941,-112.037,171.969,40.836,157.805
C06104=1043.650,294.188,-112.069,171.973,40.839,157.805
C06105=1043.657,294.436,-112.101,171.975,40.842,157.806
C06106=1043.664,294.684,-112.134,171.979,40.844,157.807
C06107=1043.671,294.932,-112.166,171.983,40.846,157.808
C06108=1043.677,295.179,-112.199,171.987,40.849,157.808
C06109=1043.684,295.427,-112.231,171.990,40.851,157.809
C06110=1043.691,295.675,-112.263,171.993,40.854,157.810
C06111=1043.698,295.923,-112.295,171.997,40.857,157.811
C06112=1043.704,296.170,-112.328,172.001,40.859,157.811
C06113=1043.710,296.418,-112.361,172.004,40.861,157.812
C06114=1043.717,296.666,-112.394,172.008,40.864,157.813
C06115=1043.724,296.914,-112.426,172.012,40.867,157.814
C06116=1043.730,297.161,-112.459,172.015,40.869,157.814
C06117=1043.737,297.409,-112.492,172.018,40.872,157.815
C06118=1043.744,297.657,-112.525,172.022,40.875,157.816
C06119=1043.751,297.904,-112.557,172.026,40.877,157.817
C06120=1043.757,298.152,-112.590,172.030,40.879,157.817
C06121=1043.763,298.399,-112.622,172.032,40.882,157.818
C06122=1043.770,298.648,-112.655,172.036,40.885,157.819
C06123=1043.776,298.895,-112.688,172.040,40.888,157.820
C06124=1043.783,299.143,-112.720,172.044,40.890,157.820
C06125=1043.790,299.391,-112.753,172.048,40.893,157.821
C06126=1043.797,299.639,-112.786,172.051,40.896,157.822
C06127=1043.803,299.886,-112.819,172.055,40.898,157.823
C06128=1043.810,300.134,-112.852,172.058,40.900,157.823
C06129=1043.817,300.382,-112.884,172.062,40.903,157.824
C06130=1043.823,300.629,-112.917,172.066,40.906,157.825
C06131=1043.830,300.878,-112.950,172.069,40.908,157.826
C06132=1043.837,301.125,-112.984,172.073,40.911,157.826
C06133=1043.843,301.372,-113.016,172.077,40.914,157.827
C06134=1043.851,301.620,-113.049,172.080,40.916,157.828
C06135=1043.857,301.868,-113.082,172.084,40.919,157.829
C06136=1043.864,302.116,-113.115,172.088,40.921,157.830
C06137=1043.870,302.363,-113.148,172.091,40.924,157.830
C06138=1043.877,302.611,-113.181,172.095,40.927,157.831
C06139=1043.884,302.859,-113.214,172.099,40.930,157.832
C06140=1043.891,303.106,-113.246,172.103,40.932,157.833
C06141=1043.898,303.354,-113.280,172.106,40.935,157.834
C06142=1043.904,303.601,-113.313,172.110,40.937,157.834
C06143=1043.911,303.850,-113.346,172.114,40.940,157.835
C06144=1043.918,304.097,-113.379,172.118,40.943,157.836
C06145=1043.924,304.345,-113.412,172.122,40.945,157.837
C06146=1043.932,304.592,-113.444,172.125,40.948,157.837
C06147=1043.940,304.897,-113.486,172.130,40.951,157.838
C06148=1043.948,305.202,-113.526,172.135,40.954,157.839
C06149=1043.957,305.507,-113.568,172.139,40.958,157.840
C06150=1043.965,305.813,-113.609,172.144,40.961,157.841
C06151=1043.972,306.060,-113.641,172.148,40.963,157.842
C06152=1043.979,306.308,-113.675,172.152,40.966,157.843
C06153=1043.986,306.555,-113.707,172.156,40.969,157.844
C06154=1043.993,306.803,-113.741,172.160,40.972,157.845
C06155=1044.000,307.051,-113.774,172.162,40.974,157.845
C06156=1044.006,307.298,-113.808,172.166,40.977,157.846
C06157=1044.014,307.546,-113.842,172.170,40.980,157.847
C06158=1044.020,307.793,-113.874,172.174,40.982,157.848
C06159=1044.027,308.041,-113.908,172.178,40.985,157.848
C06160=1044.035,308.289,-113.941,172.182,40.988,157.849
C06161=1044.041,308.536,-113.974,172.186,40.990,157.850
C06162=1044.049,308.784,-114.008,172.190,40.993,157.851
C06163=1044.055,309.032,-114.041,172.193,40.995,157.852
C06164=1044.062,309.279,-114.074,172.197,40.998,157.852
C06165=1044.069,309.527,-114.108,172.201,41.001,157.853
C06166=1044.076,309.775,-114.141,172.205,41.004,157.854
C06167=1044.083,310.022,-114.175,172.209,41.007,157.855
C06168=1044.091,310.269,-114.208,172.213,41.009,157.856
C06169=1044.098,310.518,-114.241,172.217,41.012,157.856
C06170=1044.105,310.765,-114.275,172.221,41.014,157.857
C06171=1044.111,311.012,-114.308,172.225,41.017,157.858
C06172=1044.119,311.260,-114.342,172.229,41.020,157.859
C06173=1044.126,311.508,-114.375,172.233,41.023,157.860
C06174=1044.133,311.756,-114.409,172.236,41.025,157.861
C06175=1044.140,312.021,-114.446,172.241,41.028,157.861
C06176=1044.148,312.286,-114.481,172.245,41.031,157.862
C06177=1044.155,312.552,-114.518,172.249,41.034,157.863
C06178=1044.163,312.818,-114.554,172.253,41.038,157.864
C06179=1044.169,313.065,-114.588,172.257,41.040,157.865
C06180=1044.176,313.313,-114.621,172.261,41.043,157.866
C06181=1044.183,313.560,-114.657,172.265,41.046,157.867
C06182=1044.189,313.807,-114.690,172.269,41.049,157.868
C06183=1044.196,314.055,-114.724,172.274,41.052,157.868
C06184=1044.203,314.303,-114.758,172.278,41.054,157.869
C06185=1044.209,314.551,-114.793,172.282,41.058,157.870
C06186=1044.216,314.798,-114.826,172.286,41.060,157.871
C06187=1044.223,315.046,-114.860,172.290,41.063,157.872
C06188=1044.230,315.293,-114.895,172.294,41.066,157.873
C06189=1044.237,315.541,-114.929,172.298,41.069,157.874
C06190=1044.243,315.788,-114.963,172.302,41.072,157.874
C06191=1044.250,316.036,-114.997,172.306,41.075,157.875
C06192=1044.257,316.284,-115.031,172.310,41.078,157.876
C06193=1044.264,316.531,-115.066,172.314,41.081,157.877
C06194=1044.271,316.779,-115.100,172.318,41.084,157.878
C06195=1044.277,317.026,-115.134,172.322,41.087,157.879
C06196=1044.284,317.273,-115.169,172.326,41.090,157.880
C06197=1044.291,317.521,-115.203,172.330,41.092,157.881
C06198=1044.298,317.769,-115.237,172.334,41.096,157.882
C06199=1044.305,318.016,-115.272,172.338,41.099,157.883
C06200=1044.312,318.264,-115.306,172.343,41.101,157.883
C06201=1044.319,318.511,-115.340,172.347,41.104,157.884
C06202=1044.326,318.759,-115.375,172.351,41.107,157.885
C06203=1044.334,319.086,-115.421,172.356,41.111,157.886
C06204=1044.343,319.414,-115.466,172.361,41.115,157.887
C06205=1044.353,319.742,-115.511,172.367,41.119,157.889
C06206=1044.362,320.069,-115.557,172.372,41.123,157.890
C06207=1044.369,320.316,-115.592,172.377,41.126,157.891
C06208=1044.376,320.564,-115.626,172.381,41.129,157.892
C06209=1044.383,320.811,-115.661,172.385,41.132,157.893
C06210=1044.390,321.059,-115.695,172.389,41.135,157.893
C06211=1044.397,321.307,-115.730,172.393,41.138,157.894
C06212=1044.404,321.554,-115.764,172.397,41.141,157.895
C06213=1044.411,321.802,-115.799,172.402,41.144,157.896
C06214=1044.418,322.049,-115.833,172.406,41.147,157.897
C06215=1044.425,322.297,-115.868,172.410,41.150,157.898
C06216=1044.431,322.544,-115.903,172.414,41.153,157.899
C06217=1044.439,322.792,-115.938,172.418,41.156,157.900
C06218=1044.446,323.040,-115.972,172.422,41.159,157.901
C06219=1044.453,323.287,-116.007,172.427,41.162,157.902
C06220=1044.460,323.534,-116.042,172.431,41.165,157.903
C06221=1044.467,323.782,-116.076,172.435,41.168,157.903
C06222=1044.474,324.029,-116.111,172.439,41.171,157.904
C06223=1044.481,324.277,-116.146,172.444,41.174,157.905
C06224=1044.488,324.524,-116.180,172.448,41.177,157.906
C06225=1044.496,324.772,-116.216,172.452,41.181,157.907
C06226=1044.503,325.019,-116.250,172.457,41.184,157.908
C06227=1044.510,325.267,-116.285,172.461,41.186,157.909
C06228=1044.517,325.514,-116.319,172.466,41.189,157.910
C06229=1044.524,325.761,-116.355,172.470,41.193,157.911
C06230=1044.531,326.009,-116.390,172.474,41.196,157.912
C06231=1044.539,326.256,-116.425,172.479,41.199,157.913
C06232=1044.546,326.504,-116.460,172.483,41.202,157.914
C06233=1044.553,326.751,-116.494,172.487,41.205,157.915
C06234=1044.561,326.999,-116.530,172.491,41.208,157.916
C06235=1044.567,327.246,-116.565,172.496,41.211,157.917
C06236=1044.575,327.493,-116.599,172.500,41.214,157.918
C06237=1044.582,327.740,-116.635,172.504,41.218,157.919
C06238=1044.589,327.989,-116.670,172.509,41.221,157.920
C06239=1044.596,328.236,-116.705,172.513,41.223,157.920
C06240=1044.603,328.483,-116.740,172.517,41.226,157.921
C06241=1044.611,328.731,-116.775,172.522,41.229,157.922
C06242=1044.618,328.978,-116.810,172.526,41.233,157.923
C06243=1044.625,329.225,-116.845,172.530,41.236,157.924
C06244=1044.632,329.474,-116.880,172.536,41.239,157.925
C06245=1044.639,329.721,-116.916,172.540,41.243,157.926
C06246=1044.646,329.968,-116.951,172.544,41.246,157.927
C06247=1044.653,330.216,-116.987,172.549,41.249,157.928
C06248=1044.660,330.463,-117.022,172.553,41.252,157.929
C06249=1044.667,330.710,-117.058,172.557,41.256,157.930
C06250=1044.674,330.957,-117.093,172.562,41.259,157.931
C06251=1044.681,331.205,-117.129,172.566,41.262,157.932
C06252=1044.688,331.452,-117.164,172.571,41.265,157.933
C06253=1044.695,331.699,-117.200,172.576,41.269,157.934
C06254=1044.703,331.947,-117.236,172.580,41.272,157.935
C06255=1044.710,332.194,-117.271,172.584,41.275,157.936
C06256=1044.717,332.442,-117.306,172.589,41.279,157.937
C06257=1044.724,332.689,-117.342,172.593,41.282,157.938
C06258=1044.731,332.936,-117.377,172.597,41.285,157.939
C06259=1044.741,333.259,-117.425,172.604,41.290,157.941
C06260=1044.750,333.581,-117.471,172.610,41.294,157.942
C06261=1044.760,333.905,-117.517,172.616,41.298,157.943
C06262=1044.769,334.228,-117.564,172.621,41.302,157.944
C06263=1044.776,334.474,-117.600,172.627,41.306,157.946
C06264=1044.783,334.722,-117.636,172.631,41.309,157.947
C06265=1044.790,334.969,-117.671,172.635,41.313,157.948
C06266=1044.798,335.216,-117.708,172.640,41.316,157.949
C06267=1044.805,335.465,-117.743,172.644,41.319,157.950
C06268=1044.812,335.711,-117.779,172.649,41.322,157.951
C06269=1044.820,335.959,-117.815,172.654,41.326,157.952
C06270=1044.826,336.206,-117.852,172.659,41.329,157.953
C06271=1044.834,336.454,-117.887,172.663,41.333,157.954
C06272=1044.841,336.701,-117.923,172.667,41.336,157.955
C06273=1044.848,336.948,-117.959,172.672,41.340,157.956
C06274=1044.855,337.195,-117.996,172.677,41.343,157.957
C06275=1044.862,337.443,-118.032,172.682,41.346,157.958
C06276=1044.869,337.689,-118.068,172.686,41.350,157.959
C06277=1044.876,337.937,-118.105,172.691,41.354,157.960
C06278=1044.883,338.184,-118.140,172.696,41.357,157.961
C06279=1044.891,338.431,-118.177,172.701,41.360,157.962
C06280=1044.899,338.679,-118.213,172.705,41.364,157.964
C06281=1044.905,338.926,-118.249,172.710,41.367,157.964
C06282=1044.913,339.173,-118.285,172.714,41.371,157.966
C06283=1044.920,339.420,-118.321,172.720,41.374,157.967
C06284=1044.927,339.668,-118.358,172.724,41.378,157.968
C06285=1044.934,339.915,-118.394,172.729,41.381,157.969
C06286=1044.942,340.162,-118.430,172.733,41.385,157.970
C06287=1044.948,340.410,-118.467,172.739,41.388,157.971
C06288=1044.956,340.657,-118.503,172.743,41.392,157.972
C06289=1044.964,340.905,-118.539,172.748,41.395,157.973
C06290=1044.970,341.152,-118.576,172.752,41.399,157.974
C06291=1044.978,341.398,-118.613,172.758,41.402,157.975
C06292=1044.986,341.646,-118.649,172.762,41.406,157.977
C06293=1044.992,341.893,-118.685,172.767,41.410,157.978
C06294=1045.000,342.140,-118.722,172.772,41.413,157.979
C06295=1045.007,342.387,-118.759,172.777,41.417,157.980
C06296=1045.015,342.635,-118.795,172.782,41.420,157.981
C06297=1045.021,342.882,-118.832,172.786,41.424,157.982
C06298=1045.029,343.129,-118.869,172.791,41.427,157.983
C06299=1045.036,343.377,-118.906,172.796,41.431,157.984
C06300=1045.044,343.624,-118.942,172.801,41.435,157.986
C06301=1045.051,343.871,-118.979,172.807,41.439,157.987
C06302=1045.058,344.118,-119.015,172.811,41.443,157.988
C06303=1045.065,344.365,-119.053,172.816,41.446,157.989
C06304=1045.072,344.613,-119.090,172.820,41.450,157.990
C06305=1045.080,344.860,-119.126,172.826,41.453,157.991
C06306=1045.087,345.107,-119.163,172.831,41.457,157.992
C06307=1045.094,345.353,-119.200,172.835,41.461,157.993
C06308=1045.102,345.601,-119.237,172.841,41.464,157.995
C06309=1045.109,345.848,-119.274,172.846,41.468,157.996
C06310=1045.117,346.095,-119.311,172.850,41.472,157.997
C06311=1045.124,346.342,-119.349,172.856,41.476,157.998
C06312=1045.131,346.590,-119.385,172.860,41.479,157.999
C06313=1045.139,346.837,-119.422,172.865,41.483,158.000
C06314=1045.146,347.084,-119.460,172.871,41.487,158.002
C06315=1045.155,347.403,-119.508,172.877,41.492,158.003
C06316=1045.165,347.722,-119.555,172.883,41.496,158.005
C06317=1045.174,348.041,-119.604,172.890,41.502,158.006
C06318=1045.184,348.360,-119.652,172.897,41.506,158.008
C06319=1045.192,348.607,-119.688,172.902,41.510,158.009
C06320=1045.199,348.854,-119.726,172.906,41.514,158.010
C06321=1045.206,349.101,-119.764,172.912,41.518,158.011
C06322=1045.213,349.348,-119.801,172.917,41.522,158.012
C06323=1045.221,349.595,-119.838,172.921,41.525,158.014
C06324=1045.228,349.843,-119.875,172.927,41.529,158.015
C06325=1045.236,350.090,-119.912,172.932,41.533,158.016
C06326=1045.244,350.337,-119.949,172.938,41.537,158.017
C06327=1045.251,350.583,-119.987,172.942,41.541,158.018
C06328=1045.258,350.830,-120.025,172.948,41.545,158.020
C06329=1045.266,351.078,-120.063,172.953,41.549,158.021
C06330=1045.273,351.325,-120.100,172.958,41.553,158.022
C06331=1045.280,351.572,-120.138,172.963,41.556,158.023
C06332=1045.287,351.819,-120.175,172.968,41.560,158.025
C06333=1045.295,352.067,-120.213,172.974,41.565,158.026
C06334=1045.303,352.313,-120.251,172.979,41.568,158.027
C06335=1045.310,352.560,-120.289,172.984,41.572,158.028
C06336=1045.317,352.808,-120.326,172.989,41.577,158.030
C06337=1045.324,353.055,-120.364,172.994,41.580,158.031
C06338=1045.333,353.301,-120.401,173.000,41.584,158.032
C06339=1045.340,353.548,-120.439,173.005,41.588,158.033
C06340=1045.347,353.795,-120.477,173.010,41.593,158.035
C06341=1045.355,354.042,-120.515,173.015,41.596,158.036
C06342=1045.363,354.290,-120.553,173.021,41.600,158.037
C06343=1045.370,354.536,-120.591,173.026,41.604,158.038
C06344=1045.377,354.783,-120.628,173.032,41.608,158.040
C06345=1045.385,355.030,-120.667,173.037,41.613,158.041
C06346=1045.393,355.278,-120.705,173.042,41.617,158.042
C06347=1045.400,355.524,-120.743,173.047,41.620,158.043
C06348=1045.408,355.771,-120.780,173.053,41.624,158.045
C06349=1045.416,356.018,-120.819,173.058,41.629,158.046
C06350=1045.423,356.266,-120.856,173.064,41.633,158.047
C06351=1045.431,356.512,-120.895,173.069,41.637,158.049
C06352=1045.438,356.759,-120.932,173.075,41.641,158.050
C06353=1045.446,357.006,-120.971,173.080,41.645,158.051
C06354=1045.453,357.253,-121.009,173.086,41.649,158.053
C06355=1045.461,357.500,-121.047,173.090,41.653,158.054
C06356=1045.468,357.748,-121.086,173.096,41.657,158.055
C06357=1045.476,357.994,-121.124,173.101,41.662,158.056
C06358=1045.483,358.241,-121.162,173.107,41.666,158.058
C06359=1045.491,358.488,-121.201,173.112,41.670,158.059
C06360=1045.499,358.735,-121.238,173.118,41.674,158.061
C06361=1045.506,358.982,-121.277,173.123,41.678,158.062
C06362=1045.514,359.229,-121.316,173.129,41.683,158.063
C06363=1045.521,359.476,-121.354,173.134,41.687,158.064
C06364=1045.529,359.723,-121.393,173.140,41.691,158.066
C06365=1045.537,359.969,-121.431,173.146,41.695,158.067
C06366=1045.545,360.217,-121.470,173.151,41.699,158.069
C06367=1045.552,360.463,-121.508,173.157,41.704,158.070
C06368=1045.559,360.710,-121.547,173.162,41.708,158.071
C06369=1045.568,360.957,-121.585,173.168,41.712,158.073
C06370=1045.575,361.204,-121.624,173.174,41.717,158.074
C06371=1045.585,361.528,-121.675,173.181,41.723,158.076
C06372=1045.595,361.853,-121.726,173.188,41.728,158.078
C06373=1045.606,362.178,-121.777,173.196,41.734,158.079
C06374=1045.616,362.503,-121.827,173.203,41.740,158.081
C06375=1045.623,362.749,-121.867,173.209,41.744,158.083
C06376=1045.631,362.996,-121.905,173.214,41.748,158.084
C06377=1045.638,363.243,-121.944,173.220,41.753,158.085
C06378=1045.647,363.490,-121.983,173.226,41.757,158.087
C06379=1045.653,363.736,-122.022,173.231,41.762,158.088
C06380=1045.662,363.983,-122.062,173.237,41.766,158.090
C06381=1045.669,364.230,-122.100,173.243,41.770,158.091
C06382=1045.677,364.477,-122.139,173.248,41.775,158.093
C06383=1045.685,364.724,-122.179,173.254,41.780,158.094
C06384=1045.692,364.971,-122.217,173.260,41.784,158.095
C06385=1045.700,365.217,-122.257,173.266,41.788,158.097
C06386=1045.707,365.464,-122.295,173.272,41.793,158.098
C06387=1045.715,365.711,-122.335,173.278,41.798,158.100
C06388=1045.724,365.957,-122.375,173.284,41.802,158.101
C06389=1045.730,366.204,-122.413,173.289,41.807,158.103
C06390=1045.739,366.451,-122.453,173.295,41.811,158.104
C06391=1045.747,366.698,-122.493,173.301,41.816,158.105
C06392=1045.755,366.945,-122.531,173.306,41.820,158.107
C06393=1045.762,367.191,-122.571,173.313,41.825,158.108
C06394=1045.770,367.438,-122.611,173.319,41.829,158.110
C06395=1045.778,367.685,-122.650,173.325,41.834,158.111
C06396=1045.785,367.932,-122.689,173.330,41.839,158.113
C06397=1045.793,368.178,-122.728,173.336,41.843,158.114
C06398=1045.801,368.425,-122.768,173.342,41.848,158.116
C06399=1045.809,368.672,-122.808,173.349,41.852,158.117
C06400=1045.817,368.919,-122.847,173.354,41.857,158.119
C06401=1045.826,369.165,-122.887,173.360,41.861,158.120
C06402=1045.833,369.411,-122.926,173.366,41.867,158.122
C06403=1045.841,369.658,-122.966,173.373,41.871,158.123
C06404=1045.849,369.905,-123.006,173.379,41.876,158.125
C06405=1045.857,370.152,-123.045,173.384,41.880,158.126
C06406=1045.865,370.398,-123.085,173.390,41.885,158.128
C06407=1045.873,370.645,-123.125,173.397,41.889,158.129
C06408=1045.881,370.892,-123.164,173.403,41.895,158.131
C06409=1045.889,371.139,-123.204,173.409,41.899,158.132
C06410=1045.897,371.386,-123.244,173.414,41.904,158.134
C06411=1045.904,371.633,-123.284,173.421,41.909,158.136
C06412=1045.912,371.878,-123.324,173.427,41.914,158.137
C06413=1045.920,372.125,-123.364,173.433,41.919,158.139
C06414=1045.928,372.372,-123.403,173.439,41.923,158.140
C06415=1045.936,372.619,-123.443,173.446,41.928,158.142
C06416=1045.944,372.865,-123.484,173.451,41.933,158.143
C06417=1045.952,373.112,-123.524,173.457,41.938,158.145
C06418=1045.960,373.358,-123.564,173.464,41.943,158.147
C06419=1045.967,373.605,-123.604,173.470,41.948,158.148
C06420=1045.975,373.851,-123.645,173.476,41.953,158.150
C06421=1045.983,374.098,-123.685,173.483,41.958,158.151
C06422=1045.991,374.344,-123.726,173.489,41.963,158.153
C06423=1046.000,374.591,-123.765,173.495,41.968,158.155
C06424=1046.008,374.837,-123.805,173.502,41.973,158.156
C06425=1046.015,375.084,-123.845,173.508,41.977,158.158
C06426=1046.024,375.331,-123.886,173.515,41.982,158.159
C06427=1046.035,375.675,-123.943,173.523,41.989,158.162
C06428=1046.046,376.019,-123.999,173.532,41.997,158.164
C06429=1046.057,376.363,-124.056,173.541,42.003,158.166
C06430=1046.068,376.707,-124.112,173.549,42.010,158.168
C06431=1046.076,376.953,-124.153,173.556,42.015,158.170
C06432=1046.085,377.200,-124.192,173.562,42.020,158.172
C06433=1046.093,377.446,-124.233,173.569,42.025,158.173
C06434=1046.102,377.693,-124.274,173.575,42.031,158.175
C06435=1046.110,377.940,-124.315,173.582,42.036,158.177
C06436=1046.118,378.186,-124.355,173.588,42.041,158.178
C06437=1046.126,378.432,-124.396,173.595,42.046,158.180
C06438=1046.134,378.679,-124.437,173.601,42.051,158.182
C06439=1046.142,378.925,-124.478,173.608,42.056,158.184
C06440=1046.150,379.172,-124.518,173.614,42.062,158.185
C06441=1046.159,379.419,-124.559,173.621,42.067,158.187
C06442=1046.167,379.665,-124.600,173.627,42.072,158.188
C06443=1046.174,379.912,-124.641,173.635,42.077,158.190
C06444=1046.183,380.158,-124.683,173.641,42.082,158.192
C06445=1046.191,380.404,-124.723,173.648,42.087,158.194
C06446=1046.199,380.651,-124.764,173.654,42.093,158.195
C06447=1046.207,380.898,-124.806,173.661,42.098,158.197
C06448=1046.216,381.144,-124.847,173.667,42.104,158.199
C06449=1046.224,381.390,-124.888,173.674,42.109,158.201
C06450=1046.232,381.637,-124.929,173.681,42.114,158.202
C06451=1046.240,381.883,-124.971,173.687,42.119,158.204
C06452=1046.248,382.130,-125.012,173.694,42.125,158.206
C06453=1046.257,382.375,-125.053,173.701,42.131,158.208
C06454=1046.264,382.622,-125.094,173.708,42.136,158.209
C06455=1046.273,382.868,-125.136,173.715,42.141,158.211
C06456=1046.281,383.115,-125.177,173.721,42.147,158.213
C06457=1046.290,383.361,-125.218,173.728,42.152,158.215
C06458=1046.297,383.607,-125.260,173.735,42.157,158.217
C06459=1046.306,383.854,-125.301,173.742,42.163,158.218
C06460=1046.314,384.100,-125.343,173.749,42.168,158.220
C06461=1046.323,384.346,-125.385,173.756,42.174,158.222
C06462=1046.331,384.593,-125.426,173.762,42.180,158.224
C06463=1046.340,384.839,-125.467,173.769,42.185,158.226
C06464=1046.348,385.086,-125.510,173.776,42.190,158.227
C06465=1046.356,385.331,-125.551,173.783,42.196,158.229
C06466=1046.365,385.578,-125.593,173.790,42.201,158.231
C06467=1046.374,385.825,-125.634,173.797,42.207,158.233
C06468=1046.381,386.071,-125.676,173.804,42.212,158.235
C06469=1046.390,386.317,-125.717,173.811,42.218,158.237
C06470=1046.399,386.563,-125.759,173.818,42.223,158.239
C06471=1046.407,386.809,-125.801,173.825,42.229,158.241
C06472=1046.416,387.056,-125.843,173.833,42.235,158.242
C06473=1046.425,387.302,-125.884,173.840,42.240,158.244
C06474=1046.433,387.549,-125.927,173.846,42.246,158.246
C06475=1046.441,387.794,-125.968,173.853,42.252,158.248
C06476=1046.450,388.040,-126.010,173.861,42.258,158.250
C06477=1046.459,388.287,-126.053,173.868,42.263,158.252
C06478=1046.468,388.533,-126.094,173.875,42.269,158.254
C06479=1046.476,388.780,-126.137,173.883,42.275,158.256
C06480=1046.484,389.025,-126.178,173.889,42.280,158.257
C06481=1046.493,389.272,-126.221,173.896,42.286,158.259
C06482=1046.501,389.518,-126.263,173.904,42.292,158.261
C06483=1046.515,389.895,-126.328,173.915,42.301,158.264
C06484=1046.528,390.272,-126.393,173.926,42.310,158.267
C06485=1046.541,390.649,-126.457,173.938,42.319,158.270
C06486=1046.553,391.027,-126.523,173.948,42.328,158.273
C06487=1046.563,391.273,-126.566,173.956,42.333,158.275
C06488=1046.571,391.520,-126.608,173.963,42.339,158.277
C06489=1046.580,391.766,-126.650,173.971,42.346,158.279
C06490=1046.589,392.012,-126.693,173.978,42.352,158.281
C06491=1046.597,392.258,-126.736,173.986,42.358,158.283
C06492=1046.605,392.504,-126.779,173.993,42.364,158.285
C06493=1046.615,392.750,-126.821,174.000,42.370,158.287
C06494=1046.623,392.996,-126.864,174.008,42.376,158.289
C06495=1046.632,393.242,-126.907,174.015,42.382,158.291
C06496=1046.640,393.488,-126.950,174.023,42.388,158.294
C06497=1046.649,393.734,-126.993,174.030,42.394,158.296
C06498=1046.658,393.981,-127.035,174.038,42.400,158.298
C06499=1046.666,394.227,-127.078,174.046,42.406,158.300
C06500=1046.675,394.473,-127.121,174.053,42.412,158.302
C06501=1046.683,394.718,-127.165,174.061,42.418,158.304
C06502=1046.693,394.964,-127.207,174.068,42.425,158.306
C06503=1046.701,395.210,-127.250,174.077,42.431,158.308
C06504=1046.710,395.457,-127.294,174.084,42.437,158.310
C06505=1046.719,395.703,-127.337,174.092,42.443,158.312
C06506=1046.727,395.949,-127.380,174.099,42.449,158.314
C06507=1046.737,396.194,-127.423,174.107,42.456,158.317
C06508=1046.745,396.440,-127.466,174.115,42.462,158.319
C06509=1046.754,396.687,-127.509,174.122,42.468,158.321
C06510=1046.763,396.932,-127.553,174.130,42.474,158.323
C06511=1046.772,397.178,-127.596,174.139,42.480,158.325
C06512=1046.780,397.424,-127.639,174.146,42.487,158.327
C06513=1046.790,397.670,-127.683,174.154,42.494,158.329
C06514=1046.798,397.917,-127.726,174.162,42.500,158.331
C06515=1046.807,398.162,-127.770,174.169,42.506,158.334
C06516=1046.816,398.408,-127.814,174.178,42.512,158.336
C06517=1046.825,398.654,-127.857,174.186,42.519,158.338
C06518=1046.834,398.900,-127.901,174.194,42.525,158.340
C06519=1046.843,399.146,-127.944,174.201,42.532,158.342
C06520=1046.852,399.392,-127.988,174.210,42.538,158.345
C06521=1046.861,399.638,-128.032,174.218,42.545,158.347
C06522=1046.870,399.883,-128.076,174.225,42.551,158.349
C06523=1046.879,400.130,-128.119,174.234,42.558,158.351
C06524=1046.888,400.376,-128.163,174.242,42.564,158.354
C06525=1046.896,400.622,-128.208,174.250,42.571,158.356
C06526=1046.906,400.868,-128.252,174.259,42.578,158.358
C06527=1046.915,401.114,-128.295,174.266,42.584,158.360
C06528=1046.924,401.360,-128.340,174.274,42.591,158.363
C06529=1046.933,401.605,-128.383,174.283,42.597,158.365
C06530=1046.942,401.851,-128.427,174.291,42.604,158.367
C06531=1046.952,402.097,-128.472,174.299,42.611,158.370
C06532=1046.960,402.343,-128.516,174.308,42.617,158.372
C06533=1046.969,402.589,-128.560,174.316,42.624,158.374
C06534=1046.978,402.835,-128.604,174.324,42.631,158.376
C06535=1046.987,403.081,-128.649,174.332,42.638,158.379
C06536=1046.996,403.327,-128.693,174.341,42.645,158.381
C06537=1047.006,403.573,-128.737,174.349,42.651,158.383
C06538=1047.014,403.818,-128.781,174.357,42.658,158.386
C06539=1047.030,404.215,-128.854,174.371,42.669,158.390
C06540=1047.044,404.611,-128.925,174.385,42.680,158.394
C06541=1047.059,405.007,-128.997,174.398,42.691,158.397
C06542=1047.074,405.403,-129.069,174.412,42.703,158.401
C06543=1047.083,405.649,-129.115,174.421,42.709,158.404
C06544=1047.092,405.895,-129.159,174.429,42.716,158.406
C06545=1047.101,406.141,-129.204,174.439,42.724,158.409
C06546=1047.111,406.386,-129.249,174.447,42.731,158.411
C06547=1047.119,406.633,-129.294,174.456,42.738,158.413
C06548=1047.129,406.878,-129.339,174.465,42.744,158.416
C06549=1047.138,407.124,-129.384,174.473,42.752,158.418
C06550=1047.147,407.369,-129.428,174.482,42.759,158.421
C06551=1047.157,407.615,-129.474,174.490,42.766,158.423
C06552=1047.166,407.861,-129.519,174.499,42.773,158.426
C06553=1047.175,408.107,-129.564,174.508,42.780,158.428
C06554=1047.185,408.352,-129.609,174.517,42.787,158.431
C06555=1047.194,408.598,-129.655,174.526,42.795,158.433
C06556=1047.204,408.843,-129.700,174.535,42.802,158.436
C06557=1047.213,409.089,-129.745,174.544,42.809,158.438
C06558=1047.223,409.335,-129.790,174.553,42.816,158.441
C06559=1047.232,409.581,-129.835,174.562,42.824,158.444
C06560=1047.242,409.826,-129.881,174.571,42.831,158.446
C06561=1047.251,410.072,-129.927,174.580,42.838,158.449
C06562=1047.261,410.318,-129.971,174.589,42.846,158.451
C06563=1047.270,410.563,-130.017,174.599,42.853,158.454
C06564=1047.280,410.809,-130.063,174.607,42.861,158.457
C06565=1047.289,411.055,-130.108,174.616,42.868,158.459
C06566=1047.299,411.300,-130.154,174.625,42.875,158.462
C06567=1047.309,411.546,-130.199,174.635,42.883,158.464
C06568=1047.318,411.791,-130.246,174.644,42.890,158.467
C06569=1047.328,412.037,-130.290,174.654,42.898,158.470
C06570=1047.338,412.283,-130.337,174.663,42.905,158.472
C06571=1047.348,412.528,-130.382,174.672,42.912,158.475
C06572=1047.358,412.774,-130.428,174.682,42.920,158.478
C06573=1047.367,413.019,-130.474,174.691,42.928,158.480
C06574=1047.377,413.265,-130.521,174.700,42.935,158.483
C06575=1047.386,413.511,-130.567,174.710,42.943,158.486
C06576=1047.395,413.756,-130.612,174.719,42.951,158.489
C06577=1047.406,414.002,-130.658,174.729,42.958,158.491
C06578=1047.415,414.247,-130.704,174.738,42.966,158.494
C06579=1047.425,414.493,-130.751,174.748,42.974,158.497
C06580=1047.434,414.738,-130.797,174.757,42.982,158.500
C06581=1047.444,414.984,-130.844,174.767,42.989,158.502
C06582=1047.454,415.230,-130.891,174.776,42.997,158.505
C06583=1047.463,415.475,-130.937,174.786,43.005,158.508
C06584=1047.473,415.721,-130.983,174.797,43.013,158.511
C06585=1047.483,415.966,-131.029,174.806,43.021,158.514
C06586=1047.493,416.211,-131.076,174.816,43.029,158.516
C06587=1047.503,416.457,-131.123,174.825,43.036,158.519
C06588=1047.513,416.703,-131.169,174.835,43.045,158.522
C06589=1047.523,416.947,-131.216,174.846,43.052,158.525
C06590=1047.533,417.193,-131.263,174.855,43.060,158.528
C06591=1047.543,417.438,-131.310,174.865,43.068,158.531
C06592=1047.553,417.684,-131.356,174.875,43.076,158.534
C06593=1047.563,417.930,-131.403,174.885,43.084,158.537
C06594=1047.572,418.175,-131.450,174.895,43.092,158.539
C06595=1047.589,418.579,-131.527,174.912,43.106,158.544
C06596=1047.606,418.981,-131.604,174.928,43.119,158.549
C06597=1047.623,419.385,-131.682,174.945,43.132,158.554
C06598=1047.639,419.788,-131.760,174.962,43.146,158.559
C06599=1047.649,420.034,-131.807,174.972,43.154,158.562
C06600=1047.659,420.279,-131.854,174.983,43.162,158.565
C06601=1047.669,420.524,-131.902,174.993,43.171,158.568
C06602=1047.679,420.769,-131.949,175.003,43.179,158.571
C06603=1047.689,421.015,-131.997,175.013,43.187,158.574
C06604=1047.699,421.260,-132.044,175.024,43.196,158.577
C06605=1047.709,421.506,-132.091,175.034,43.204,158.580
C06606=1047.720,421.750,-132.139,175.045,43.213,158.583
C06607=1047.730,421.996,-132.186,175.056,43.221,158.586
C06608=1047.739,422.241,-132.234,175.066,43.230,158.590
C06609=1047.751,422.486,-132.282,175.077,43.238,158.593
C06610=1047.761,422.732,-132.330,175.087,43.247,158.596
C06611=1047.771,422.976,-132.377,175.098,43.255,158.599
C06612=1047.781,423.222,-132.425,175.109,43.264,158.602
C06613=1047.792,423.467,-132.474,175.121,43.272,158.605
C06614=1047.802,423.712,-132.521,175.130,43.281,158.608
C06615=1047.812,423.957,-132.569,175.142,43.289,158.611
C06616=1047.824,424.203,-132.617,175.153,43.298,158.615
C06617=1047.833,424.448,-132.666,175.164,43.307,158.618
C06618=1047.843,424.693,-132.713,175.174,43.316,158.621
C06619=1047.855,424.938,-132.761,175.185,43.324,158.624
C06620=1047.865,425.183,-132.809,175.196,43.333,158.628
C06621=1047.875,425.429,-132.858,175.208,43.342,158.631
C06622=1047.886,425.673,-132.906,175.219,43.351,158.634
C06623=1047.896,425.919,-132.955,175.230,43.360,158.638
C06624=1047.907,426.164,-133.003,175.242,43.369,158.641
C06625=1047.917,426.409,-133.052,175.252,43.377,158.644
C06626=1047.928,426.653,-133.100,175.263,43.386,158.648
C06627=1047.938,426.899,-133.149,175.275,43.396,158.651
C06628=1047.949,427.144,-133.197,175.286,43.405,158.654
C06629=1047.960,427.389,-133.247,175.297,43.414,158.658
C06630=1047.970,427.633,-133.295,175.309,43.422,158.661
C06631=1047.981,427.878,-133.344,175.320,43.432,158.664
C06632=1047.992,428.124,-133.392,175.333,43.441,158.668
C06633=1048.003,428.368,-133.441,175.344,43.450,158.671
C06634=1048.013,428.614,-133.490,175.356,43.459,158.675
C06635=1048.024,428.858,-133.539,175.367,43.468,158.678
C06636=1048.035,429.104,-133.588,175.379,43.477,158.682
C06637=1048.045,429.349,-133.637,175.390,43.486,158.685
C06638=1048.056,429.593,-133.686,175.402,43.496,158.689
C06639=1048.067,429.838,-133.736,175.414,43.505,158.692
C06640=1048.078,430.083,-133.785,175.426,43.514,158.696
C06641=1048.088,430.328,-133.835,175.438,43.524,158.699
C06642=1048.100,430.573,-133.884,175.449,43.533,158.703
C06643=1048.110,430.818,-133.934,175.462,43.543,158.706
C06644=1048.120,431.062,-133.983,175.474,43.552,158.710
C06645=1048.132,431.307,-134.032,175.485,43.562,158.714
C06646=1048.143,431.552,-134.082,175.498,43.571,158.717
C06647=1048.153,431.797,-134.132,175.510,43.580,158.721
C06648=1048.164,432.042,-134.181,175.522,43.590,158.724
C06649=1048.176,432.286,-134.231,175.534,43.600,158.728
C06650=1048.186,432.531,-134.281,175.546,43.609,158.732
C06651=1048.196,432.745,-134.324,175.557,43.618,158.735
C06652=1048.206,432.957,-134.368,175.569,43.626,158.738
C06653=1048.216,433.171,-134.411,175.579,43.635,158.742
C06654=1048.225,433.384,-134.454,175.590,43.643,158.745
C06655=1048.235,433.597,-134.499,175.600,43.652,158.748
C06656=1048.245,433.810,-134.542,175.612,43.660,158.751
C06657=1048.255,434.024,-134.585,175.622,43.669,158.755
C06658=1048.264,434.236,-134.629,175.633,43.677,158.758
C06659=1048.276,434.481,-134.680,175.646,43.687,158.762
C06660=1048.287,434.726,-134.730,175.658,43.697,158.765
C06661=1048.298,434.970,-134.780,175.671,43.706,158.769
C06662=1048.309,435.216,-134.830,175.684,43.716,158.773
C06663=1048.321,435.460,-134.880,175.698,43.726,158.777
C06664=1048.332,435.705,-134.931,175.710,43.736,158.781
C06665=1048.344,435.949,-134.982,175.723,43.746,158.785
C06666=1048.355,436.194,-135.032,175.736,43.756,158.789
C06667=1048.366,436.438,-135.083,175.749,43.766,158.792
C06668=1048.378,436.684,-135.133,175.762,43.776,158.796
C06669=1048.389,436.927,-135.184,175.776,43.787,158.800
C06670=1048.401,437.173,-135.235,175.789,43.797,158.804
C06671=1048.412,437.416,-135.286,175.802,43.807,158.808
C06672=1048.423,437.661,-135.337,175.815,43.817,158.812
C06673=1048.435,437.907,-135.388,175.829,43.828,158.816
C06674=1048.447,438.151,-135.439,175.842,43.838,158.821
C06675=1048.459,438.396,-135.490,175.855,43.848,158.825
C06676=1048.470,438.641,-135.541,175.869,43.859,158.829
C06677=1048.482,438.885,-135.592,175.882,43.869,158.833
C06678=1048.493,439.129,-135.644,175.896,43.880,158.837
C06679=1048.505,439.374,-135.695,175.909,43.890,158.841
C06680=1048.516,439.618,-135.746,175.923,43.901,158.845
C06681=1048.528,439.862,-135.798,175.937,43.911,158.849
C06682=1048.540,440.107,-135.849,175.951,43.921,158.853
C06683=1048.552,440.351,-135.901,175.964,43.932,158.858
C06684=1048.564,440.595,-135.953,175.978,43.943,158.862
C06685=1048.576,440.840,-136.004,175.993,43.953,158.866
C06686=1048.587,441.084,-136.056,176.007,43.964,158.871
C06687=1048.599,441.328,-136.108,176.020,43.975,158.875
C06688=1048.611,441.573,-136.160,176.035,43.985,158.879
C06689=1048.623,441.817,-136.212,176.049,43.996,158.883
C06690=1048.635,442.061,-136.263,176.063,44.007,158.888
C06691=1048.646,442.305,-136.316,176.077,44.018,158.892
C06692=1048.659,442.549,-136.368,176.092,44.029,158.896
C06693=1048.670,442.794,-136.420,176.106,44.040,158.901
C06694=1048.683,443.038,-136.472,176.121,44.050,158.905
C06695=1048.694,443.282,-136.524,176.136,44.061,158.910
C06696=1048.707,443.527,-136.577,176.150,44.073,158.914
C06697=1048.719,443.770,-136.629,176.165,44.084,158.919
C06698=1048.730,444.015,-136.682,176.180,44.095,158.923
C06699=1048.743,444.258,-136.734,176.194,44.106,158.928
C06700=1048.755,444.503,-136.786,176.209,44.117,158.932
C06701=1048.768,444.746,-136.839,176.224,44.128,158.937
C06702=1048.779,444.991,-136.892,176.239,44.140,158.941
C06703=1048.792,445.235,-136.945,176.254,44.150,158.946
C06704=1048.805,445.478,-136.997,176.268,44.162,158.950
C06705=1048.817,445.722,-137.050,176.284,44.173,158.955
C06706=1048.829,445.966,-137.102,176.299,44.185,158.960
C06707=1048.843,446.208,-137.154,176.314,44.195,158.964
C06708=1048.857,446.451,-137.205,176.330,44.207,158.969
C06709=1048.872,446.695,-137.257,176.345,44.217,158.973
C06710=1048.888,446.939,-137.306,176.360,44.228,158.978
C06711=1048.901,447.159,-137.352,176.375,44.237,158.982
C06712=1048.917,447.378,-137.396,176.389,44.247,158.986
C06713=1048.932,447.598,-137.440,176.403,44.256,158.990
C06714=1048.948,447.817,-137.484,176.417,44.265,158.994
C06715=1048.965,448.037,-137.528,176.431,44.275,158.998
C06716=1048.982,448.258,-137.570,176.446,44.283,159.001
C06717=1049.000,448.478,-137.613,176.460,44.292,159.005
C06718=1049.019,448.700,-137.655,176.474,44.300,159.009
C06719=1049.039,448.944,-137.701,176.491,44.310,159.014
C06720=1049.061,449.189,-137.745,176.507,44.320,159.018
C06721=1049.084,449.434,-137.791,176.523,44.329,159.022
C06722=1049.106,449.679,-137.836,176.540,44.338,159.026
C06723=1049.130,449.924,-137.880,176.556,44.347,159.030
C06724=1049.156,450.170,-137.924,176.572,44.355,159.034
C06725=1049.181,450.415,-137.966,176.589,44.364,159.039
C06726=1049.207,450.660,-138.009,176.605,44.373,159.043
C06727=1048.895,450.691,-138.311,176.606,44.463,159.069
C06728=1048.869,450.445,-138.269,176.590,44.454,159.065
C06729=1048.843,450.200,-138.226,176.572,44.446,159.061
C06730=1048.819,449.954,-138.183,176.556,44.437,159.057
C06731=1048.795,449.709,-138.139,176.539,44.428,159.052
C06732=1048.772,449.464,-138.094,176.523,44.419,159.048
C06733=1048.749,449.219,-138.049,176.507,44.410,159.044
C06734=1048.727,448.974,-138.004,176.491,44.401,159.040
C06735=1048.706,448.729,-137.958,176.474,44.391,159.036
C06736=1048.688,448.518,-137.917,176.460,44.383,159.032
C06737=1048.671,448.306,-137.877,176.446,44.375,159.028
C06738=1048.654,448.094,-137.836,176.433,44.366,159.024
C06739=1048.638,447.883,-137.794,176.419,44.358,159.021
C06740=1048.622,447.672,-137.753,176.405,44.349,159.017
C06741=1048.606,447.461,-137.710,176.392,44.340,159.013
C06742=1048.592,447.250,-137.669,176.378,44.332,159.009
C06743=1048.578,447.040,-137.625,176.365,44.322,159.005
C06744=1048.562,446.796,-137.575,176.349,44.312,159.001
C06745=1048.547,446.552,-137.524,176.334,44.301,158.996
C06746=1048.532,446.308,-137.473,176.317,44.290,158.992
C06747=1048.518,446.066,-137.422,176.302,44.280,158.987
C06748=1048.506,445.822,-137.370,176.287,44.268,158.983
C06749=1048.493,445.579,-137.317,176.272,44.258,158.978
C06750=1048.481,445.335,-137.264,176.257,44.246,158.973
C06751=1048.468,445.092,-137.211,176.241,44.235,158.969
C06752=1048.456,444.848,-137.159,176.227,44.224,158.964
C06753=1048.443,444.604,-137.107,176.212,44.212,158.960
C06754=1048.431,444.360,-137.054,176.197,44.202,158.955
C06755=1048.419,444.115,-137.001,176.182,44.191,158.951
C06756=1048.407,443.872,-136.949,176.167,44.179,158.946
C06757=1048.394,443.628,-136.896,176.153,44.168,158.942
C06758=1048.382,443.383,-136.843,176.138,44.157,158.937
C06759=1048.370,443.139,-136.791,176.123,44.146,158.933
C06760=1048.358,442.895,-136.739,176.109,44.136,158.928
C06761=1048.346,442.651,-136.687,176.094,44.125,158.924
C06762=1048.335,442.406,-136.635,176.079,44.114,158.919
C06763=1048.322,442.162,-136.583,176.065,44.103,158.915
C06764=1048.310,441.919,-136.531,176.050,44.093,158.911
C06765=1048.298,441.673,-136.479,176.037,44.082,158.906
C06766=1048.286,441.429,-136.426,176.022,44.071,158.902
C06767=1048.274,441.185,-136.375,176.008,44.060,158.898
C06768=1048.262,440.941,-136.323,175.994,44.050,158.894
C06769=1048.250,440.696,-136.271,175.980,44.039,158.889
C06770=1048.239,440.452,-136.220,175.966,44.029,158.885
C06771=1048.227,440.208,-136.168,175.951,44.018,158.881
C06772=1048.215,439.964,-136.117,175.938,44.007,158.877
C06773=1048.203,439.719,-136.065,175.924,43.997,158.873
C06774=1048.191,439.475,-136.014,175.911,43.987,158.868
C06775=1048.180,439.230,-135.962,175.896,43.976,158.864
C06776=1048.168,438.986,-135.911,175.883,43.966,158.860
C06777=1048.157,438.742,-135.860,175.869,43.955,158.856
C06778=1048.145,438.497,-135.808,175.856,43.945,158.852
C06779=1048.133,438.253,-135.757,175.842,43.935,158.848
C06780=1048.122,438.008,-135.706,175.829,43.925,158.844
C06781=1048.110,437.764,-135.655,175.816,43.914,158.840
C06782=1048.098,437.519,-135.604,175.802,43.904,158.836
C06783=1048.088,437.275,-135.553,175.789,43.894,158.832
C06784=1048.076,437.030,-135.502,175.775,43.884,158.828
C06785=1048.065,436.786,-135.452,175.762,43.874,158.824
C06786=1048.053,436.541,-135.400,175.749,43.864,158.820
C06787=1048.042,436.297,-135.350,175.736,43.854,158.816
C06788=1048.030,436.052,-135.299,175.723,43.844,158.812
C06789=1048.019,435.808,-135.249,175.709,43.834,158.808
C06790=1048.007,435.563,-135.199,175.696,43.824,158.804
C06791=1047.996,435.319,-135.148,175.684,43.814,158.800
C06792=1047.984,435.074,-135.097,175.671,43.804,158.796
C06793=1047.973,434.829,-135.047,175.658,43.795,158.792
C06794=1047.962,434.585,-134.998,175.645,43.785,158.789
C06795=1047.950,434.339,-134.947,175.633,43.775,158.785
C06796=1047.941,434.125,-134.903,175.622,43.766,158.782
C06797=1047.930,433.911,-134.859,175.610,43.758,158.778
C06798=1047.921,433.696,-134.815,175.600,43.749,158.775
C06799=1047.911,433.482,-134.771,175.588,43.741,158.772
C06800=1047.901,433.268,-134.727,175.577,43.732,158.768
C06801=1047.891,433.054,-134.683,175.567,43.724,158.765
C06802=1047.882,432.838,-134.640,175.556,43.715,158.762
C06803=1047.872,432.625,-134.596,175.544,43.707,158.758
C06804=1047.861,432.380,-134.546,175.532,43.698,158.755
C06805=1047.850,432.135,-134.496,175.520,43.688,158.751
C06806=1047.839,431.890,-134.447,175.508,43.678,158.747
C06807=1047.828,431.646,-134.397,175.495,43.669,158.744
C06808=1047.818,431.424,-134.351,175.485,43.660,158.741
C06809=1047.808,431.202,-134.307,175.473,43.652,158.737
C06810=1047.798,430.981,-134.262,175.462,43.644,158.734
C06811=1047.788,430.759,-134.217,175.452,43.635,158.731
C06812=1047.778,430.537,-134.173,175.441,43.626,158.728
C06813=1047.769,430.316,-134.128,175.429,43.618,158.724
C06814=1047.759,430.094,-134.083,175.419,43.609,158.721
C06815=1047.750,429.872,-134.038,175.408,43.601,158.718
C06816=1047.738,429.627,-133.989,175.396,43.592,158.714
C06817=1047.728,429.382,-133.940,175.385,43.582,158.711
C06818=1047.717,429.137,-133.890,175.373,43.573,158.707
C06819=1047.706,428.892,-133.841,175.360,43.564,158.704
C06820=1047.695,428.647,-133.792,175.349,43.555,158.700
C06821=1047.685,428.402,-133.744,175.337,43.546,158.697
C06822=1047.674,428.157,-133.694,175.326,43.537,158.694
C06823=1047.663,427.912,-133.646,175.315,43.528,158.690
C06824=1047.653,427.668,-133.597,175.303,43.519,158.687
C06825=1047.642,427.422,-133.548,175.292,43.510,158.683
C06826=1047.630,427.177,-133.499,175.280,43.501,158.680
C06827=1047.620,426.933,-133.451,175.269,43.492,158.677
C06828=1047.609,426.687,-133.402,175.258,43.483,158.673
C06829=1047.599,426.443,-133.353,175.246,43.474,158.670
C06830=1047.588,426.197,-133.305,175.235,43.465,158.666
C06831=1047.578,425.952,-133.256,175.224,43.457,158.663
C06832=1047.567,425.707,-133.208,175.212,43.448,158.660
C06833=1047.558,425.462,-133.160,175.201,43.439,158.657
C06834=1047.546,425.217,-133.111,175.190,43.430,158.653
C06835=1047.536,424.972,-133.063,175.178,43.421,158.650
C06836=1047.526,424.726,-133.014,175.167,43.413,158.647
C06837=1047.515,424.482,-132.966,175.156,43.404,158.644
C06838=1047.505,424.237,-132.919,175.146,43.396,158.640
C06839=1047.494,423.992,-132.870,175.135,43.387,158.637
C06840=1047.484,423.746,-132.822,175.124,43.378,158.634
C06841=1047.473,423.501,-132.774,175.112,43.370,158.631
C06842=1047.462,423.256,-132.726,175.102,43.361,158.628
C06843=1047.452,423.011,-132.679,175.091,43.352,158.624
C06844=1047.442,422.766,-132.631,175.080,43.344,158.621
C06845=1047.432,422.520,-132.583,175.069,43.336,158.618
C06846=1047.421,422.275,-132.535,175.059,43.327,158.615
C06847=1047.411,422.030,-132.488,175.048,43.319,158.612
C06848=1047.401,421.785,-132.441,175.038,43.310,158.609
C06849=1047.390,421.540,-132.393,175.027,43.302,158.606
C06850=1047.381,421.294,-132.345,175.016,43.294,158.603
C06851=1047.370,421.048,-132.297,175.006,43.285,158.600
C06852=1047.360,420.803,-132.250,174.995,43.277,158.597
C06853=1047.349,420.558,-132.202,174.985,43.269,158.594
C06854=1047.339,420.313,-132.155,174.974,43.261,158.590
C06855=1047.330,420.068,-132.107,174.964,43.253,158.587
C06856=1047.320,419.842,-132.064,174.955,43.245,158.585
C06857=1047.311,419.616,-132.021,174.945,43.237,158.582
C06858=1047.302,419.391,-131.977,174.936,43.230,158.579
C06859=1047.292,419.164,-131.933,174.926,43.222,158.576
C06860=1047.283,418.939,-131.890,174.917,43.215,158.574
C06861=1047.275,418.713,-131.847,174.907,43.207,158.571
C06862=1047.265,418.486,-131.803,174.898,43.200,158.568
C06863=1047.255,418.260,-131.760,174.888,43.193,158.566
C06864=1047.245,418.015,-131.713,174.878,43.185,158.563
C06865=1047.235,417.769,-131.666,174.869,43.176,158.560
C06866=1047.226,417.525,-131.620,174.858,43.169,158.557
C06867=1047.216,417.279,-131.573,174.848,43.161,158.554
C06868=1047.206,417.033,-131.526,174.839,43.153,158.551
C06869=1047.196,416.788,-131.479,174.829,43.145,158.548
C06870=1047.186,416.542,-131.432,174.818,43.137,158.545
C06871=1047.176,416.297,-131.387,174.809,43.129,158.542
C06872=1047.166,416.051,-131.340,174.799,43.121,158.540
C06873=1047.156,415.806,-131.293,174.789,43.113,158.537
C06874=1047.146,415.561,-131.247,174.779,43.106,158.534
C06875=1047.136,415.315,-131.200,174.769,43.098,158.531
C06876=1047.126,415.069,-131.154,174.760,43.090,158.528
C06877=1047.117,414.824,-131.108,174.750,43.082,158.526
C06878=1047.107,414.578,-131.061,174.740,43.074,158.523
C06879=1047.097,414.334,-131.015,174.731,43.067,158.520
C06880=1047.087,414.088,-130.968,174.721,43.059,158.517
C06881=1047.078,413.843,-130.922,174.712,43.051,158.515
C06882=1047.068,413.597,-130.876,174.703,43.044,158.512
C06883=1047.059,413.351,-130.830,174.693,43.036,158.509
C06884=1047.049,413.105,-130.784,174.683,43.029,158.506
C06885=1047.040,412.860,-130.738,174.674,43.021,158.504
C06886=1047.029,412.614,-130.692,174.665,43.013,158.501
C06887=1047.020,412.369,-130.646,174.655,43.006,158.498
C06888=1047.010,412.122,-130.600,174.646,42.999,158.496
C06889=1047.000,411.878,-130.554,174.637,42.992,158.493
C06890=1046.991,411.632,-130.509,174.627,42.984,158.490
C06891=1046.981,411.386,-130.463,174.618,42.976,158.488
C06892=1046.972,411.140,-130.418,174.608,42.969,158.485
C06893=1046.962,410.895,-130.372,174.599,42.962,158.482
C06894=1046.952,410.649,-130.326,174.590,42.954,158.480
C06895=1046.942,410.404,-130.281,174.580,42.947,158.477
C06896=1046.933,410.158,-130.235,174.571,42.940,158.475
C06897=1046.923,409.912,-130.190,174.562,42.933,158.472
C06898=1046.914,409.666,-130.145,174.554,42.926,158.470
C06899=1046.904,409.421,-130.099,174.545,42.918,158.467
C06900=1046.895,409.175,-130.054,174.535,42.911,158.464
C06901=1046.885,408.930,-130.009,174.526,42.904,158.462
C06902=1046.876,408.683,-129.963,174.517,42.897,158.459
C06903=1046.866,408.438,-129.918,174.509,42.889,158.457
C06904=1046.857,408.192,-129.873,174.500,42.882,158.454
C06905=1046.847,407.947,-129.828,174.490,42.875,158.452
C06906=1046.838,407.701,-129.783,174.481,42.868,158.449
C06907=1046.828,407.455,-129.738,174.473,42.861,158.447
C06908=1046.819,407.209,-129.692,174.464,42.854,158.444
C06909=1046.810,406.964,-129.648,174.455,42.847,158.442
C06910=1046.801,406.718,-129.602,174.447,42.840,158.439
C06911=1046.791,406.473,-129.557,174.437,42.833,158.437
C06912=1046.782,406.226,-129.513,174.428,42.826,158.434
C06913=1046.773,405.981,-129.468,174.420,42.819,158.432
C06914=1046.764,405.735,-129.422,174.411,42.812,158.429
C06915=1046.754,405.489,-129.378,174.403,42.805,158.427
C06916=1046.740,405.091,-129.306,174.389,42.794,158.423
C06917=1046.725,404.693,-129.233,174.375,42.782,158.419
C06918=1046.710,404.295,-129.161,174.362,42.772,158.415
C06919=1046.696,403.896,-129.088,174.348,42.760,158.411
C06920=1046.686,403.650,-129.044,174.339,42.754,158.409
C06921=1046.677,403.404,-128.999,174.331,42.747,158.407
C06922=1046.668,403.159,-128.956,174.322,42.740,158.404
C06923=1046.659,402.913,-128.910,174.314,42.734,158.402
C06924=1046.649,402.667,-128.866,174.305,42.727,158.400
C06925=1046.641,402.421,-128.822,174.297,42.720,158.397
C06926=1046.631,402.175,-128.778,174.289,42.713,158.395
C06927=1046.622,401.929,-128.734,174.280,42.707,158.393
C06928=1046.614,401.683,-128.690,174.272,42.700,158.390
C06929=1046.604,401.437,-128.646,174.264,42.694,158.388
C06930=1046.595,401.191,-128.602,174.256,42.687,158.386
C06931=1046.586,400.946,-128.558,174.248,42.681,158.384
C06932=1046.577,400.700,-128.514,174.239,42.674,158.381
C06933=1046.568,400.454,-128.470,174.231,42.667,158.379
C06934=1046.559,400.208,-128.425,174.222,42.661,158.377
C06935=1046.550,399.962,-128.382,174.215,42.654,158.375
C06936=1046.541,399.716,-128.338,174.207,42.648,158.372
C06937=1046.532,399.470,-128.295,174.199,42.641,158.370
C06938=1046.523,399.224,-128.250,174.190,42.635,158.368
C06939=1046.514,398.979,-128.207,174.183,42.629,158.366
C06940=1046.505,398.732,-128.163,174.175,42.622,158.364
C06941=1046.496,398.486,-128.120,174.166,42.616,158.361
C06942=1046.487,398.241,-128.076,174.159,42.610,158.359
C06943=1046.478,397.994,-128.032,174.151,42.603,158.357
C06944=1046.470,397.749,-127.989,174.143,42.597,158.355
C06945=1046.460,397.502,-127.945,174.134,42.590,158.353
C06946=1046.452,397.257,-127.902,174.127,42.584,158.351
C06947=1046.442,397.011,-127.859,174.119,42.578,158.348
C06948=1046.434,396.765,-127.815,174.111,42.571,158.346
C06949=1046.425,396.519,-127.772,174.104,42.565,158.344
C06950=1046.416,396.273,-127.729,174.095,42.559,158.342
C06951=1046.407,396.027,-127.685,174.087,42.553,158.340
C06952=1046.399,395.781,-127.642,174.080,42.547,158.338
C06953=1046.390,395.534,-127.599,174.072,42.541,158.336
C06954=1046.381,395.288,-127.556,174.065,42.535,158.334
C06955=1046.372,395.043,-127.512,174.057,42.528,158.331
C06956=1046.363,394.797,-127.470,174.049,42.522,158.329
C06957=1046.355,394.551,-127.427,174.042,42.516,158.327
C06958=1046.345,394.304,-127.383,174.033,42.510,158.325
C06959=1046.337,394.058,-127.340,174.026,42.504,158.323
C06960=1046.328,393.812,-127.297,174.018,42.498,158.321
C06961=1046.319,393.566,-127.255,174.011,42.492,158.319
C06962=1046.311,393.320,-127.212,174.003,42.486,158.317
C06963=1046.302,393.074,-127.169,173.996,42.480,158.315
C06964=1046.294,392.828,-127.126,173.988,42.474,158.313
C06965=1046.285,392.582,-127.084,173.981,42.468,158.311
C06966=1046.276,392.336,-127.041,173.973,42.462,158.309
C06967=1046.268,392.090,-126.998,173.966,42.456,158.307
C06968=1046.259,391.844,-126.955,173.958,42.450,158.305
C06969=1046.250,391.597,-126.913,173.951,42.444,158.303
C06970=1046.242,391.351,-126.870,173.943,42.438,158.301
C06971=1046.233,391.106,-126.828,173.936,42.432,158.299
C06972=1046.220,390.726,-126.763,173.925,42.423,158.296
C06973=1046.206,390.346,-126.697,173.913,42.414,158.293
C06974=1046.194,389.968,-126.632,173.902,42.406,158.290
C06975=1046.180,389.588,-126.566,173.891,42.397,158.287
C06976=1046.171,389.342,-126.524,173.884,42.391,158.285
C06977=1046.163,389.096,-126.481,173.876,42.385,158.283
C06978=1046.155,388.849,-126.439,173.869,42.379,158.281
C06979=1046.146,388.604,-126.398,173.861,42.374,158.279
C06980=1046.138,388.357,-126.356,173.854,42.368,158.277
C06981=1046.129,388.111,-126.313,173.848,42.362,158.275
C06982=1046.120,387.865,-126.271,173.840,42.356,158.273
C06983=1046.111,387.618,-126.230,173.833,42.351,158.271
C06984=1046.104,387.372,-126.188,173.826,42.345,158.269
C06985=1046.095,387.126,-126.146,173.819,42.340,158.268
C06986=1046.086,386.880,-126.104,173.811,42.335,158.266
C06987=1046.078,386.633,-126.062,173.805,42.329,158.264
C06988=1046.069,386.387,-126.021,173.798,42.323,158.262
C06989=1046.060,386.141,-125.979,173.791,42.318,158.260
C06990=1046.052,385.894,-125.937,173.783,42.312,158.258
C06991=1046.044,385.649,-125.895,173.776,42.307,158.256
C06992=1046.035,385.402,-125.854,173.770,42.301,158.255
C06993=1046.027,385.156,-125.811,173.763,42.296,158.253
C06994=1046.019,384.909,-125.771,173.755,42.290,158.251
C06995=1046.010,384.663,-125.729,173.748,42.285,158.249
C06996=1046.001,384.416,-125.687,173.742,42.279,158.247
C06997=1045.993,384.171,-125.645,173.735,42.274,158.245
C06998=1045.984,383.924,-125.604,173.728,42.269,158.244
C06999=1045.976,383.678,-125.563,173.721,42.263,158.242
C07000=1045.968,383.431,-125.521,173.714,42.257,158.240
C07001=1045.960,383.185,-125.480,173.707,42.252,158.238
C07002=1045.951,382.939,-125.438,173.701,42.247,158.237
C07003=1045.944,382.692,-125.397,173.694,42.241,158.235
C07004=1045.935,382.446,-125.355,173.687,42.236,158.233
C07005=1045.927,382.199,-125.315,173.680,42.231,158.231
C07006=1045.918,381.953,-125.273,173.673,42.225,158.229
C07007=1045.911,381.706,-125.232,173.666,42.220,158.228
C07008=1045.902,381.461,-125.190,173.660,42.215,158.226
C07009=1045.894,381.214,-125.149,173.653,42.210,158.224
C07010=1045.885,380.968,-125.108,173.647,42.204,158.222
C07011=1045.877,380.721,-125.066,173.640,42.199,158.221
C07012=1045.869,380.475,-125.026,173.633,42.194,158.219
C07013=1045.861,380.229,-124.984,173.626,42.188,158.217
C07014=1045.853,379.982,-124.943,173.619,42.183,158.215
C07015=1045.845,379.735,-124.902,173.613,42.178,158.214
C07016=1045.837,379.489,-124.861,173.606,42.173,158.212
C07017=1045.829,379.243,-124.821,173.600,42.167,158.210
C07018=1045.820,378.996,-124.780,173.593,42.163,158.209
C07019=1045.812,378.750,-124.739,173.587,42.157,158.207
C07020=1045.804,378.503,-124.699,173.580,42.152,158.205
C07021=1045.796,378.256,-124.658,173.574,42.147,158.204
C07022=1045.788,378.010,-124.617,173.567,42.142,158.202
C07023=1045.780,377.764,-124.576,173.561,42.137,158.200
C07024=1045.771,377.517,-124.535,173.554,42.132,158.199
C07025=1045.763,377.270,-124.495,173.548,42.127,158.197
C07026=1045.755,377.024,-124.454,173.541,42.122,158.195
C07027=1045.747,376.778,-124.413,173.535,42.117,158.194
C07028=1045.735,376.432,-124.357,173.525,42.110,158.191
C07029=1045.724,376.086,-124.300,173.516,42.103,158.189
C07030=1045.712,375.740,-124.243,173.508,42.096,158.187
C07031=1045.701,375.394,-124.186,173.499,42.089,158.184
C07032=1045.693,375.147,-124.147,173.492,42.084,158.183
C07033=1045.685,374.901,-124.106,173.486,42.079,158.181
C07034=1045.677,374.654,-124.065,173.480,42.074,158.180
C07035=1045.669,374.407,-124.025,173.473,42.069,158.178
C07036=1045.661,374.161,-123.985,173.467,42.065,158.176
C07037=1045.653,373.914,-123.945,173.460,42.060,158.175
C07038=1045.645,373.668,-123.905,173.455,42.055,158.173
C07039=1045.637,373.421,-123.865,173.449,42.050,158.172
C07040=1045.629,373.175,-123.824,173.442,42.045,158.170
C07041=1045.621,372.928,-123.784,173.436,42.040,158.168
C07042=1045.613,372.682,-123.744,173.430,42.035,158.167
C07043=1045.606,372.435,-123.704,173.423,42.031,158.165
C07044=1045.598,372.188,-123.664,173.417,42.026,158.164
C07045=1045.589,371.942,-123.624,173.411,42.021,158.162
C07046=1045.581,371.695,-123.584,173.405,42.016,158.161
C07047=1045.574,371.448,-123.544,173.398,42.011,158.159
C07048=1045.566,371.201,-123.504,173.393,42.007,158.157
C07049=1045.558,370.955,-123.463,173.387,42.002,158.156
C07050=1045.550,370.708,-123.423,173.380,41.997,158.154
C07051=1045.542,370.461,-123.384,173.374,41.993,158.153
C07052=1045.534,370.215,-123.344,173.368,41.988,158.151
C07053=1045.526,369.968,-123.305,173.363,41.983,158.150
C07054=1045.518,369.721,-123.265,173.356,41.979,158.148
C07055=1045.510,369.475,-123.226,173.350,41.974,158.147
C07056=1045.502,369.228,-123.186,173.344,41.970,158.145
C07057=1045.494,368.982,-123.147,173.339,41.965,158.144
C07058=1045.486,368.735,-123.107,173.332,41.961,158.142
C07059=1045.478,368.488,-123.067,173.326,41.955,158.141
C07060=1045.470,368.241,-123.028,173.320,41.951,158.139
C07061=1045.463,367.994,-122.989,173.314,41.947,158.138
C07062=1045.455,367.748,-122.949,173.309,41.942,158.136
C07063=1045.447,367.501,-122.910,173.302,41.938,158.135
C07064=1045.439,367.254,-122.870,173.296,41.933,158.134
C07065=1045.432,367.008,-122.831,173.290,41.928,158.132
C07066=1045.423,366.761,-122.792,173.285,41.924,158.131
C07067=1045.416,366.514,-122.752,173.279,41.919,158.129
C07068=1045.407,366.267,-122.714,173.272,41.915,158.128
C07069=1045.400,366.021,-122.674,173.267,41.911,158.126
C07070=1045.392,365.774,-122.635,173.261,41.906,158.125
C07071=1045.384,365.526,-122.595,173.255,41.901,158.123
C07072=1045.377,365.281,-122.556,173.249,41.897,158.122
C07073=1045.369,365.033,-122.517,173.244,41.893,158.120
C07074=1045.361,364.786,-122.478,173.238,41.888,158.119
C07075=1045.354,364.540,-122.439,173.232,41.883,158.118
C07076=1045.346,364.293,-122.399,173.226,41.879,158.116
C07077=1045.339,364.046,-122.361,173.220,41.875,158.115
C07078=1045.331,363.799,-122.321,173.214,41.870,158.113
C07079=1045.323,363.553,-122.283,173.209,41.866,158.112
C07080=1045.315,363.306,-122.243,173.203,41.861,158.110
C07081=1045.307,363.059,-122.204,173.197,41.857,158.109
C07082=1045.300,362.812,-122.166,173.191,41.853,158.108
C07083=1045.292,362.565,-122.126,173.186,41.848,158.106
C07084=1045.282,362.239,-122.075,173.179,41.842,158.104
C07085=1045.272,361.912,-122.024,173.170,41.837,158.103
C07086=1045.262,361.585,-121.973,173.163,41.831,158.101
C07087=1045.252,361.259,-121.922,173.156,41.826,158.099
C07088=1045.244,361.012,-121.883,173.151,41.821,158.098
C07089=1045.236,360.765,-121.845,173.145,41.817,158.096
C07090=1045.229,360.518,-121.806,173.139,41.813,158.095
C07091=1045.221,360.271,-121.767,173.134,41.809,158.094
C07092=1045.213,360.025,-121.729,173.128,41.805,158.092
C07093=1045.205,359.777,-121.691,173.123,41.800,158.091
C07094=1045.198,359.531,-121.652,173.117,41.796,158.089
C07095=1045.190,359.283,-121.613,173.111,41.792,158.088
C07096=1045.183,359.037,-121.575,173.106,41.788,158.087
C07097=1045.175,358.790,-121.537,173.100,41.784,158.085
C07098=1045.167,358.543,-121.498,173.095,41.779,158.084
C07099=1045.159,358.297,-121.460,173.089,41.775,158.083
C07100=1045.151,358.049,-121.421,173.084,41.771,158.082
C07101=1045.145,357.802,-121.383,173.078,41.767,158.080
C07102=1045.137,357.556,-121.345,173.073,41.763,158.079
C07103=1045.129,357.308,-121.306,173.067,41.758,158.077
C07104=1045.122,357.062,-121.268,173.061,41.754,158.076
C07105=1045.114,356.815,-121.230,173.056,41.750,158.075
C07106=1045.106,356.567,-121.192,173.052,41.747,158.074
C07107=1045.099,356.320,-121.154,173.046,41.742,158.072
C07108=1045.091,356.074,-121.116,173.040,41.738,158.071
C07109=1045.084,355.827,-121.078,173.035,41.734,158.070
C07110=1045.076,355.579,-121.040,173.029,41.730,158.068
C07111=1045.068,355.333,-121.002,173.024,41.726,158.067
C07112=1045.061,355.086,-120.964,173.018,41.722,158.066
C07113=1045.054,354.839,-120.926,173.013,41.718,158.065
C07114=1045.046,354.591,-120.888,173.008,41.714,158.063
C07115=1045.038,354.345,-120.850,173.003,41.710,158.062
C07116=1045.031,354.098,-120.812,172.997,41.706,158.061
C07117=1045.024,353.851,-120.775,172.992,41.702,158.060
C07118=1045.016,353.603,-120.736,172.987,41.698,158.058
C07119=1045.008,353.356,-120.699,172.981,41.694,158.057
C07120=1045.001,353.109,-120.661,172.976,41.691,158.056
C07121=1044.994,352.863,-120.623,172.971,41.686,158.055
C07122=1044.986,352.616,-120.585,172.966,41.682,158.053
C07123=1044.979,352.368,-120.548,172.960,41.679,158.052
C07124=1044.971,352.122,-120.510,172.955,41.675,158.051
C07125=1044.964,351.875,-120.473,172.949,41.671,158.050
C07126=1044.956,351.627,-120.435,172.945,41.667,158.048
C07127=1044.948,351.380,-120.397,172.939,41.663,158.047
C07128=1044.941,351.133,-120.360,172.934,41.659,158.046
C07129=1044.934,350.886,-120.322,172.929,41.655,158.045
C07130=1044.926,350.639,-120.284,172.924,41.651,158.043
C07131=1044.919,350.392,-120.246,172.919,41.647,158.042
C07132=1044.912,350.145,-120.209,172.913,41.644,158.041
C07133=1044.904,349.898,-120.172,172.908,41.640,158.040
C07134=1044.897,349.651,-120.134,172.904,41.636,158.039
C07135=1044.889,349.404,-120.097,172.898,41.632,158.037
C07136=1044.881,349.157,-120.060,172.893,41.628,158.036
C07137=1044.874,348.910,-120.022,172.887,41.625,158.035
C07138=1044.867,348.662,-119.986,172.883,41.621,158.034
C07139=1044.860,348.415,-119.948,172.878,41.617,158.033
C07140=1044.850,348.094,-119.900,172.871,41.612,158.031
C07141=1044.840,347.774,-119.851,172.864,41.608,158.030
C07142=1044.830,347.453,-119.803,172.857,41.603,158.028
C07143=1044.821,347.132,-119.755,172.852,41.598,158.027
C07144=1044.814,346.885,-119.718,172.846,41.594,158.025
C07145=1044.807,346.637,-119.681,172.841,41.590,158.024
C07146=1044.799,346.391,-119.644,172.837,41.586,158.023
C07147=1044.792,346.143,-119.606,172.831,41.583,158.022
C07148=1044.785,345.896,-119.570,172.826,41.579,158.021
C07149=1044.777,345.649,-119.533,172.822,41.576,158.020
C07150=1044.770,345.402,-119.495,172.816,41.572,158.018
C07151=1044.762,345.154,-119.459,172.811,41.569,158.017
C07152=1044.755,344.907,-119.421,172.807,41.565,158.016
C07153=1044.748,344.660,-119.385,172.801,41.561,158.015
C07154=1044.740,344.413,-119.348,172.797,41.557,158.014
C07155=1044.733,344.166,-119.311,172.792,41.553,158.013
C07156=1044.725,343.919,-119.274,172.786,41.550,158.011
C07157=1044.719,343.671,-119.237,172.782,41.546,158.010
C07158=1044.711,343.425,-119.201,172.777,41.543,158.009
C07159=1044.704,343.177,-119.164,172.771,41.540,158.008
C07160=1044.697,342.930,-119.127,172.767,41.536,158.007
C07161=1044.689,342.682,-119.090,172.762,41.532,158.006
C07162=1044.683,342.435,-119.054,172.758,41.529,158.005
C07163=1044.675,342.189,-119.017,172.752,41.525,158.004
C07164=1044.668,341.941,-118.980,172.748,41.521,158.003
C07165=1044.660,341.693,-118.944,172.743,41.518,158.001
C07166=1044.653,341.447,-118.908,172.737,41.514,158.000
C07167=1044.646,341.200,-118.871,172.733,41.511,157.999
C07168=1044.638,340.952,-118.834,172.728,41.508,157.998
C07169=1044.631,340.705,-118.798,172.724,41.504,157.997
C07170=1044.624,340.458,-118.762,172.718,41.500,157.996
C07171=1044.617,340.210,-118.725,172.714,41.497,157.995
C07172=1044.609,339.963,-118.689,172.709,41.494,157.994
C07173=1044.603,339.716,-118.653,172.705,41.490,157.993
C07174=1044.595,339.468,-118.617,172.700,41.487,157.992
C07175=1044.587,339.221,-118.580,172.695,41.483,157.991
C07176=1044.580,338.975,-118.544,172.690,41.480,157.989
C07177=1044.573,338.727,-118.507,172.686,41.476,157.989
C07178=1044.565,338.479,-118.471,172.681,41.473,157.987
C07179=1044.559,338.232,-118.436,172.676,41.469,157.986
C07180=1044.552,337.984,-118.399,172.671,41.466,157.985
C07181=1044.545,337.738,-118.363,172.667,41.462,157.984
C07182=1044.537,337.490,-118.327,172.662,41.459,157.983
C07183=1044.531,337.243,-118.290,172.657,41.456,157.982
C07184=1044.523,336.996,-118.254,172.652,41.452,157.981
C07185=1044.515,336.748,-118.218,172.648,41.449,157.980
C07186=1044.508,336.501,-118.182,172.643,41.445,157.979
C07187=1044.501,336.254,-118.145,172.639,41.442,157.978
C07188=1044.494,336.006,-118.110,172.633,41.439,157.977
C07189=1044.487,335.759,-118.074,172.629,41.435,157.976
C07190=1044.480,335.512,-118.038,172.624,41.432,157.975
C07191=1044.472,335.265,-118.002,172.620,41.429,157.974
C07192=1044.466,335.017,-117.966,172.616,41.426,157.973
C07193=1044.458,334.770,-117.930,172.610,41.422,157.972
C07194=1044.451,334.523,-117.894,172.606,41.419,157.971
C07195=1044.444,334.275,-117.859,172.601,41.415,157.969
C07196=1044.434,333.950,-117.812,172.596,41.411,157.968
C07197=1044.425,333.626,-117.765,172.589,41.407,157.967
C07198=1044.416,333.302,-117.718,172.584,41.403,157.966
C07199=1044.406,332.977,-117.672,172.577,41.398,157.964
C07200=1044.398,332.729,-117.635,172.573,41.395,157.963
C07201=1044.392,332.482,-117.600,172.569,41.392,157.962
C07202=1044.384,332.235,-117.564,172.564,41.389,157.961
C07203=1044.377,331.987,-117.529,172.559,41.385,157.960
C07204=1044.370,331.740,-117.493,172.554,41.382,157.959
C07205=1044.363,331.492,-117.457,172.550,41.379,157.958
C07206=1044.357,331.245,-117.422,172.546,41.376,157.957
C07207=1044.350,330.998,-117.386,172.541,41.372,157.956
C07208=1044.342,330.750,-117.350,172.537,41.369,157.955
C07209=1044.335,330.503,-117.315,172.533,41.366,157.954
C07210=1044.328,330.256,-117.279,172.528,41.363,157.953
C07211=1044.321,330.008,-117.244,172.523,41.360,157.952
C07212=1044.314,329.760,-117.209,172.519,41.356,157.951
C07213=1044.307,329.514,-117.173,172.514,41.353,157.950
C07214=1044.300,329.266,-117.138,172.510,41.350,157.949
C07215=1044.292,329.019,-117.103,172.506,41.346,157.948
C07216=1044.285,328.771,-117.068,172.501,41.343,157.947
C07217=1044.278,328.524,-117.033,172.497,41.341,157.946
